REGION Network 9: fDoor5 monitoring
   RUNG wire#powerrail
      Contact( #TRUE )
      wire#w1
      Contact( "Safety.DataFromSafety".fDoorCoilStatus.weightNgBoxDoorUnlock )
      wire#w2
      Coil( "SafetyDoorInterface".fDoor5Interface.monitoring.DoorOpen )
   END_RUNG
   RUNG wire#w1
      I_Contact( "Safety.DataFromSafety".fDoorCoilStatus.weightNgBoxDoorUnlock )
      Contact( "Safety.DataFromSafety".fDoorDrive.fDoor5.ackReq )
      I_Contact( "Global.Data".general.clock.cycle1000Msec )
      I_Contact( "Safety.DataFromSafety".fDoorSwitchStatus.weightNgBoxDoorOpen )
   END_RUNG wire#w2
   RUNG wire#w1
      Contact( "Safety.DataFromSafety".fDoorCoilStatus.weightNgBoxDoorUnlock )
      Coil( "SafetyDoorInterface".fDoor5Interface.monitoring.DoorUnLock )
   END_RUNG
   RUNG wire#w1
      I_Contact( "Safety.DataFromSafety".fDoorCoilStatus.weightNgBoxDoorUnlock )
      wire#w3
      I_Contact( "Safety.DataFromSafety".fDoorDrive.fDoor5.ackReq )
      wire#w4
      I_Contact( "Safety.DataFromSafety".fDoorSwitchStatus.weightNgBoxDoorOpen )
      I_Contact( "SafetyDoorInterface".fDoor5Interface.monitoring.DoorOpen )
      Coil( "SafetyDoorInterface".fDoor5Interface.monitoring.DoorClose )
   END_RUNG
   RUNG wire#w3
      Contact( "Safety.DataFromSafety".fDoorDrive.fDoor5.ackReq )
      I_Contact( "Global.Data".general.clock.cycle1000Msec )
   END_RUNG wire#w4
   RUNG wire#w4
      Coil( "SafetyDoorInterface".fDoor5Interface.monitoring.DoorLock )
   END_RUNG
   // the same network as SCL:
   "SafetyDoorInterface".fDoor5Interface.monitoring.DoorOpen := #TRUE AND ("Safety.DataFromSafety".fDoorCoilStatus.weightNgBoxDoorUnlock OR (NOT "Safety.DataFromSafety".fDoorCoilStatus.weightNgBoxDoorUnlock AND "Safety.DataFromSafety".fDoorDrive.fDoor5.ackReq AND NOT "Global.Data".general.clock.cycle1000Msec AND NOT "Safety.DataFromSafety".fDoorSwitchStatus.weightNgBoxDoorOpen));
   "SafetyDoorInterface".fDoor5Interface.monitoring.DoorUnLock := #TRUE AND "Safety.DataFromSafety".fDoorCoilStatus.weightNgBoxDoorUnlock;
   #_w1 := #TRUE AND NOT "Safety.DataFromSafety".fDoorCoilStatus.weightNgBoxDoorUnlock AND (NOT "Safety.DataFromSafety".fDoorDrive.fDoor5.ackReq OR ("Safety.DataFromSafety".fDoorDrive.fDoor5.ackReq AND NOT "Global.Data".general.clock.cycle1000Msec));
   "SafetyDoorInterface".fDoor5Interface.monitoring.DoorClose := #_w1 AND NOT "Safety.DataFromSafety".fDoorSwitchStatus.weightNgBoxDoorOpen AND NOT "SafetyDoorInterface".fDoor5Interface.monitoring.DoorOpen;
   "SafetyDoorInterface".fDoor5Interface.monitoring.DoorLock := #_w1;
END_REGION

REGION Network 10: fDoor5 Command
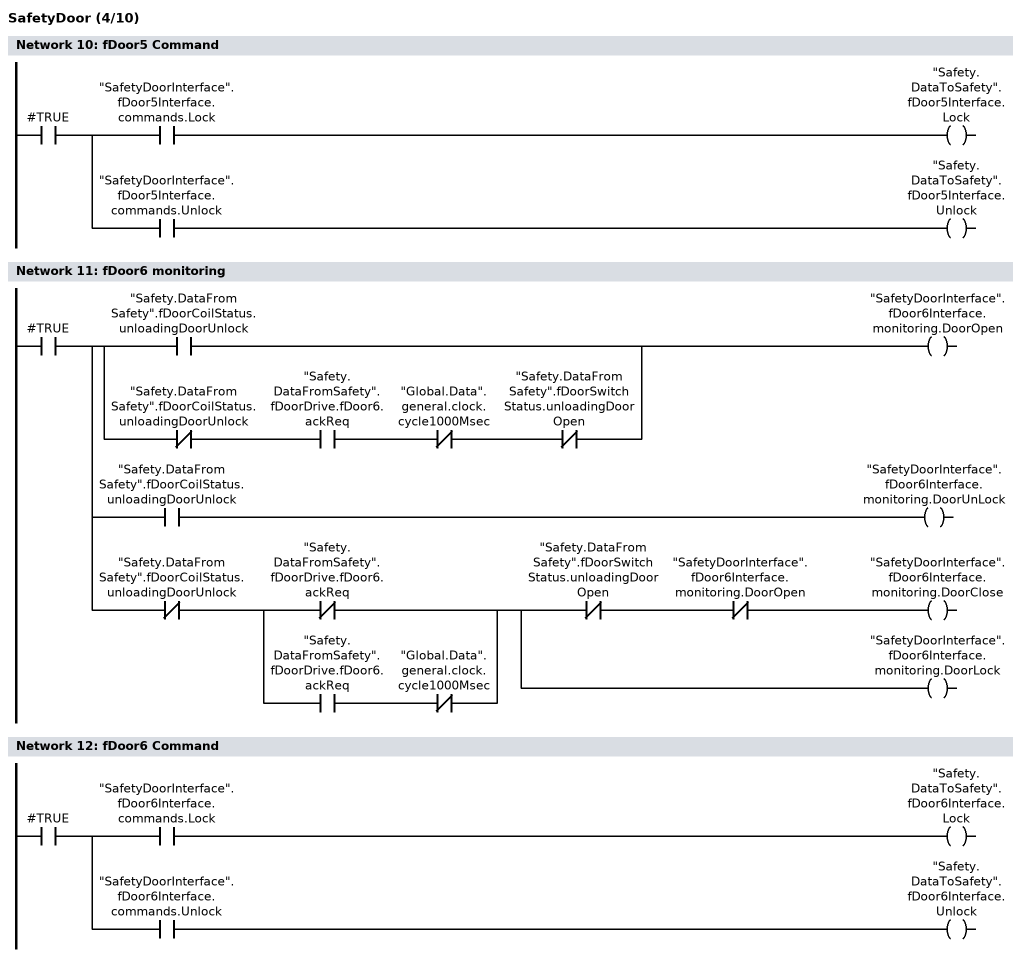
   RUNG wire#powerrail
      Contact( #TRUE )
      wire#w1
      Contact( "SafetyDoorInterface".fDoor5Interface.commands.Lock )
      Coil( "Safety.DataToSafety".fDoor5Interface.Lock )
   END_RUNG
   RUNG wire#w1
      Contact( "SafetyDoorInterface".fDoor5Interface.commands.Unlock )
      Coil( "Safety.DataToSafety".fDoor5Interface.Unlock )
   END_RUNG
   // the same network as SCL:
   "Safety.DataToSafety".fDoor5Interface.Lock := #TRUE AND "SafetyDoorInterface".fDoor5Interface.commands.Lock;
   "Safety.DataToSafety".fDoor5Interface.Unlock := #TRUE AND "SafetyDoorInterface".fDoor5Interface.commands.Unlock;
END_REGION

REGION Network 11: fDoor6 monitoring
   RUNG wire#powerrail
      Contact( #TRUE )
      wire#w1
      Contact( "Safety.DataFromSafety".fDoorCoilStatus.unloadingDoorUnlock )
      wire#w2
      Coil( "SafetyDoorInterface".fDoor6Interface.monitoring.DoorOpen )
   END_RUNG
   RUNG wire#w1
      I_Contact( "Safety.DataFromSafety".fDoorCoilStatus.unloadingDoorUnlock )
      Contact( "Safety.DataFromSafety".fDoorDrive.fDoor6.ackReq )
      I_Contact( "Global.Data".general.clock.cycle1000Msec )
      I_Contact( "Safety.DataFromSafety".fDoorSwitchStatus.unloadingDoorOpen )
   END_RUNG wire#w2
   RUNG wire#w1
      Contact( "Safety.DataFromSafety".fDoorCoilStatus.unloadingDoorUnlock )
      Coil( "SafetyDoorInterface".fDoor6Interface.monitoring.DoorUnLock )
   END_RUNG
   RUNG wire#w1
      I_Contact( "Safety.DataFromSafety".fDoorCoilStatus.unloadingDoorUnlock )
      wire#w3
      I_Contact( "Safety.DataFromSafety".fDoorDrive.fDoor6.ackReq )
      wire#w4
      I_Contact( "Safety.DataFromSafety".fDoorSwitchStatus.unloadingDoorOpen )
      I_Contact( "SafetyDoorInterface".fDoor6Interface.monitoring.DoorOpen )
      Coil( "SafetyDoorInterface".fDoor6Interface.monitoring.DoorClose )
   END_RUNG
   RUNG wire#w3
      Contact( "Safety.DataFromSafety".fDoorDrive.fDoor6.ackReq )
      I_Contact( "Global.Data".general.clock.cycle1000Msec )
   END_RUNG wire#w4
   RUNG wire#w4
      Coil( "SafetyDoorInterface".fDoor6Interface.monitoring.DoorLock )
   END_RUNG
   // the same network as SCL:
   "SafetyDoorInterface".fDoor6Interface.monitoring.DoorOpen := #TRUE AND ("Safety.DataFromSafety".fDoorCoilStatus.unloadingDoorUnlock OR (NOT "Safety.DataFromSafety".fDoorCoilStatus.unloadingDoorUnlock AND "Safety.DataFromSafety".fDoorDrive.fDoor6.ackReq AND NOT "Global.Data".general.clock.cycle1000Msec AND NOT "Safety.DataFromSafety".fDoorSwitchStatus.unloadingDoorOpen));
   "SafetyDoorInterface".fDoor6Interface.monitoring.DoorUnLock := #TRUE AND "Safety.DataFromSafety".fDoorCoilStatus.unloadingDoorUnlock;
   #_w1 := #TRUE AND NOT "Safety.DataFromSafety".fDoorCoilStatus.unloadingDoorUnlock AND (NOT "Safety.DataFromSafety".fDoorDrive.fDoor6.ackReq OR ("Safety.DataFromSafety".fDoorDrive.fDoor6.ackReq AND NOT "Global.Data".general.clock.cycle1000Msec));
   "SafetyDoorInterface".fDoor6Interface.monitoring.DoorClose := #_w1 AND NOT "Safety.DataFromSafety".fDoorSwitchStatus.unloadingDoorOpen AND NOT "SafetyDoorInterface".fDoor6Interface.monitoring.DoorOpen;
   "SafetyDoorInterface".fDoor6Interface.monitoring.DoorLock := #_w1;
END_REGION

REGION Network 12: fDoor6 Command
   RUNG wire#powerrail
      Contact( #TRUE )
      wire#w1
      Contact( "SafetyDoorInterface".fDoor6Interface.commands.Lock )
      Coil( "Safety.DataToSafety".fDoor6Interface.Lock )
   END_RUNG
   RUNG wire#w1
      Contact( "SafetyDoorInterface".fDoor6Interface.commands.Unlock )
      Coil( "Safety.DataToSafety".fDoor6Interface.Unlock )
   END_RUNG
   // the same network as SCL:
   "Safety.DataToSafety".fDoor6Interface.Lock := #TRUE AND "SafetyDoorInterface".fDoor6Interface.commands.Lock;
   "Safety.DataToSafety".fDoor6Interface.Unlock := #TRUE AND "SafetyDoorInterface".fDoor6Interface.commands.Unlock;
END_REGION

REGION Network 13: fDoor7 monitoring
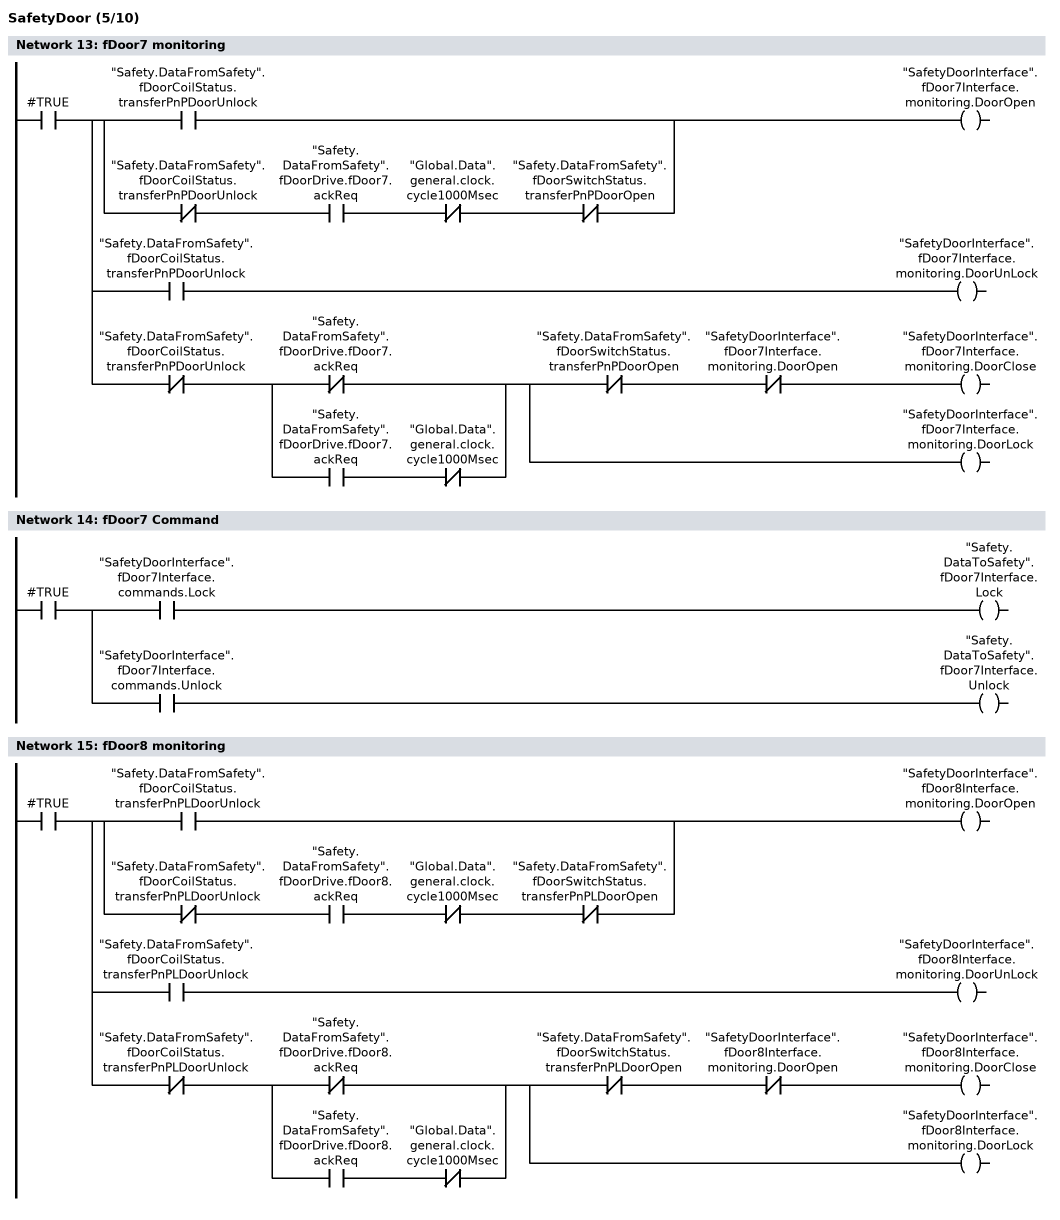
   RUNG wire#powerrail
      Contact( #TRUE )
      wire#w1
      Contact( "Safety.DataFromSafety".fDoorCoilStatus.transferPnPDoorUnlock )
      wire#w2
      Coil( "SafetyDoorInterface".fDoor7Interface.monitoring.DoorOpen )
   END_RUNG
   RUNG wire#w1
      I_Contact( "Safety.DataFromSafety".fDoorCoilStatus.transferPnPDoorUnlock )
      Contact( "Safety.DataFromSafety".fDoorDrive.fDoor7.ackReq )
      I_Contact( "Global.Data".general.clock.cycle1000Msec )
      I_Contact( "Safety.DataFromSafety".fDoorSwitchStatus.transferPnPDoorOpen )
   END_RUNG wire#w2
   RUNG wire#w1
      Contact( "Safety.DataFromSafety".fDoorCoilStatus.transferPnPDoorUnlock )
      Coil( "SafetyDoorInterface".fDoor7Interface.monitoring.DoorUnLock )
   END_RUNG
   RUNG wire#w1
      I_Contact( "Safety.DataFromSafety".fDoorCoilStatus.transferPnPDoorUnlock )
      wire#w3
      I_Contact( "Safety.DataFromSafety".fDoorDrive.fDoor7.ackReq )
      wire#w4
      I_Contact( "Safety.DataFromSafety".fDoorSwitchStatus.transferPnPDoorOpen )
      I_Contact( "SafetyDoorInterface".fDoor7Interface.monitoring.DoorOpen )
      Coil( "SafetyDoorInterface".fDoor7Interface.monitoring.DoorClose )
   END_RUNG
   RUNG wire#w3
      Contact( "Safety.DataFromSafety".fDoorDrive.fDoor7.ackReq )
      I_Contact( "Global.Data".general.clock.cycle1000Msec )
   END_RUNG wire#w4
   RUNG wire#w4
      Coil( "SafetyDoorInterface".fDoor7Interface.monitoring.DoorLock )
   END_RUNG
   // the same network as SCL:
   "SafetyDoorInterface".fDoor7Interface.monitoring.DoorOpen := #TRUE AND ("Safety.DataFromSafety".fDoorCoilStatus.transferPnPDoorUnlock OR (NOT "Safety.DataFromSafety".fDoorCoilStatus.transferPnPDoorUnlock AND "Safety.DataFromSafety".fDoorDrive.fDoor7.ackReq AND NOT "Global.Data".general.clock.cycle1000Msec AND NOT "Safety.DataFromSafety".fDoorSwitchStatus.transferPnPDoorOpen));
   "SafetyDoorInterface".fDoor7Interface.monitoring.DoorUnLock := #TRUE AND "Safety.DataFromSafety".fDoorCoilStatus.transferPnPDoorUnlock;
   #_w1 := #TRUE AND NOT "Safety.DataFromSafety".fDoorCoilStatus.transferPnPDoorUnlock AND (NOT "Safety.DataFromSafety".fDoorDrive.fDoor7.ackReq OR ("Safety.DataFromSafety".fDoorDrive.fDoor7.ackReq AND NOT "Global.Data".general.clock.cycle1000Msec));
   "SafetyDoorInterface".fDoor7Interface.monitoring.DoorClose := #_w1 AND NOT "Safety.DataFromSafety".fDoorSwitchStatus.transferPnPDoorOpen AND NOT "SafetyDoorInterface".fDoor7Interface.monitoring.DoorOpen;
   "SafetyDoorInterface".fDoor7Interface.monitoring.DoorLock := #_w1;
END_REGION

REGION Network 14: fDoor7 Command
   RUNG wire#powerrail
      Contact( #TRUE )
      wire#w1
      Contact( "SafetyDoorInterface".fDoor7Interface.commands.Lock )
      Coil( "Safety.DataToSafety".fDoor7Interface.Lock )
   END_RUNG
   RUNG wire#w1
      Contact( "SafetyDoorInterface".fDoor7Interface.commands.Unlock )
      Coil( "Safety.DataToSafety".fDoor7Interface.Unlock )
   END_RUNG
   // the same network as SCL:
   "Safety.DataToSafety".fDoor7Interface.Lock := #TRUE AND "SafetyDoorInterface".fDoor7Interface.commands.Lock;
   "Safety.DataToSafety".fDoor7Interface.Unlock := #TRUE AND "SafetyDoorInterface".fDoor7Interface.commands.Unlock;
END_REGION

REGION Network 15: fDoor8 monitoring
   RUNG wire#powerrail
      Contact( #TRUE )
      wire#w1
      Contact( "Safety.DataFromSafety".fDoorCoilStatus.transferPnPLDoorUnlock )
      wire#w2
      Coil( "SafetyDoorInterface".fDoor8Interface.monitoring.DoorOpen )
   END_RUNG
   RUNG wire#w1
      I_Contact( "Safety.DataFromSafety".fDoorCoilStatus.transferPnPLDoorUnlock )
      Contact( "Safety.DataFromSafety".fDoorDrive.fDoor8.ackReq )
      I_Contact( "Global.Data".general.clock.cycle1000Msec )
      I_Contact( "Safety.DataFromSafety".fDoorSwitchStatus.transferPnPLDoorOpen )
   END_RUNG wire#w2
   RUNG wire#w1
      Contact( "Safety.DataFromSafety".fDoorCoilStatus.transferPnPLDoorUnlock )
      Coil( "SafetyDoorInterface".fDoor8Interface.monitoring.DoorUnLock )
   END_RUNG
   RUNG wire#w1
      I_Contact( "Safety.DataFromSafety".fDoorCoilStatus.transferPnPLDoorUnlock )
      wire#w3
      I_Contact( "Safety.DataFromSafety".fDoorDrive.fDoor8.ackReq )
      wire#w4
      I_Contact( "Safety.DataFromSafety".fDoorSwitchStatus.transferPnPLDoorOpen )
      I_Contact( "SafetyDoorInterface".fDoor8Interface.monitoring.DoorOpen )
      Coil( "SafetyDoorInterface".fDoor8Interface.monitoring.DoorClose )
   END_RUNG
   RUNG wire#w3
      Contact( "Safety.DataFromSafety".fDoorDrive.fDoor8.ackReq )
      I_Contact( "Global.Data".general.clock.cycle1000Msec )
   END_RUNG wire#w4
   RUNG wire#w4
      Coil( "SafetyDoorInterface".fDoor8Interface.monitoring.DoorLock )
   END_RUNG
   // the same network as SCL:
   "SafetyDoorInterface".fDoor8Interface.monitoring.DoorOpen := #TRUE AND ("Safety.DataFromSafety".fDoorCoilStatus.transferPnPLDoorUnlock OR (NOT "Safety.DataFromSafety".fDoorCoilStatus.transferPnPLDoorUnlock AND "Safety.DataFromSafety".fDoorDrive.fDoor8.ackReq AND NOT "Global.Data".general.clock.cycle1000Msec AND NOT "Safety.DataFromSafety".fDoorSwitchStatus.transferPnPLDoorOpen));
   "SafetyDoorInterface".fDoor8Interface.monitoring.DoorUnLock := #TRUE AND "Safety.DataFromSafety".fDoorCoilStatus.transferPnPLDoorUnlock;
   #_w1 := #TRUE AND NOT "Safety.DataFromSafety".fDoorCoilStatus.transferPnPLDoorUnlock AND (NOT "Safety.DataFromSafety".fDoorDrive.fDoor8.ackReq OR ("Safety.DataFromSafety".fDoorDrive.fDoor8.ackReq AND NOT "Global.Data".general.clock.cycle1000Msec));
   "SafetyDoorInterface".fDoor8Interface.monitoring.DoorClose := #_w1 AND NOT "Safety.DataFromSafety".fDoorSwitchStatus.transferPnPLDoorOpen AND NOT "SafetyDoorInterface".fDoor8Interface.monitoring.DoorOpen;
   "SafetyDoorInterface".fDoor8Interface.monitoring.DoorLock := #_w1;
END_REGION

REGION Network 16: fDoor8 Command
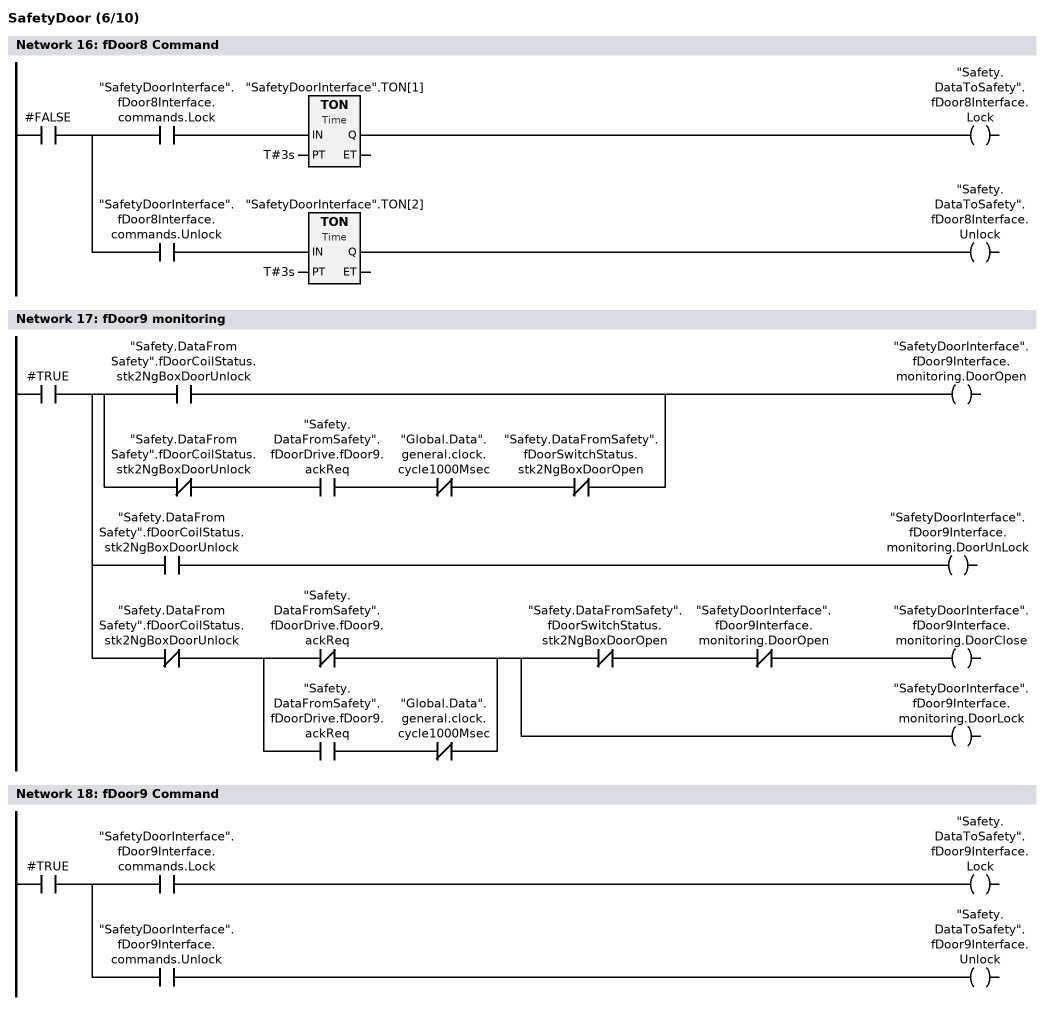
   RUNG wire#powerrail
      Contact( #FALSE )
      wire#w1
      Contact( "SafetyDoorInterface".fDoor8Interface.commands.Lock )
      { S7_Templates := "time_type := Time" } "SafetyDoorInterface".TON[1].TON(pt := T#3s, et =>)
      Coil( "Safety.DataToSafety".fDoor8Interface.Lock )
   END_RUNG
   RUNG wire#w1
      Contact( "SafetyDoorInterface".fDoor8Interface.commands.Unlock )
      { S7_Templates := "time_type := Time" } "SafetyDoorInterface".TON[2].TON(pt := T#3s, et =>)
      Coil( "Safety.DataToSafety".fDoor8Interface.Unlock )
   END_RUNG
   // the same network as SCL:
   "SafetyDoorInterface".TON[1].TON(IN := #FALSE AND "SafetyDoorInterface".fDoor8Interface.commands.Lock,
                           PT := T#3s);
   "Safety.DataToSafety".fDoor8Interface.Lock := "SafetyDoorInterface".TON[1].Q;
   "SafetyDoorInterface".TON[2].TON(IN := #FALSE AND "SafetyDoorInterface".fDoor8Interface.commands.Unlock,
                           PT := T#3s);
   "Safety.DataToSafety".fDoor8Interface.Unlock := "SafetyDoorInterface".TON[2].Q;
END_REGION

REGION Network 17: fDoor9 monitoring
   RUNG wire#powerrail
      Contact( #TRUE )
      wire#w1
      Contact( "Safety.DataFromSafety".fDoorCoilStatus.stk2NgBoxDoorUnlock )
      wire#w2
      Coil( "SafetyDoorInterface".fDoor9Interface.monitoring.DoorOpen )
   END_RUNG
   RUNG wire#w1
      I_Contact( "Safety.DataFromSafety".fDoorCoilStatus.stk2NgBoxDoorUnlock )
      Contact( "Safety.DataFromSafety".fDoorDrive.fDoor9.ackReq )
      I_Contact( "Global.Data".general.clock.cycle1000Msec )
      I_Contact( "Safety.DataFromSafety".fDoorSwitchStatus.stk2NgBoxDoorOpen )
   END_RUNG wire#w2
   RUNG wire#w1
      Contact( "Safety.DataFromSafety".fDoorCoilStatus.stk2NgBoxDoorUnlock )
      Coil( "SafetyDoorInterface".fDoor9Interface.monitoring.DoorUnLock )
   END_RUNG
   RUNG wire#w1
      I_Contact( "Safety.DataFromSafety".fDoorCoilStatus.stk2NgBoxDoorUnlock )
      wire#w3
      I_Contact( "Safety.DataFromSafety".fDoorDrive.fDoor9.ackReq )
      wire#w4
      I_Contact( "Safety.DataFromSafety".fDoorSwitchStatus.stk2NgBoxDoorOpen )
      I_Contact( "SafetyDoorInterface".fDoor9Interface.monitoring.DoorOpen )
      Coil( "SafetyDoorInterface".fDoor9Interface.monitoring.DoorClose )
   END_RUNG
   RUNG wire#w3
      Contact( "Safety.DataFromSafety".fDoorDrive.fDoor9.ackReq )
      I_Contact( "Global.Data".general.clock.cycle1000Msec )
   END_RUNG wire#w4
   RUNG wire#w4
      Coil( "SafetyDoorInterface".fDoor9Interface.monitoring.DoorLock )
   END_RUNG
   // the same network as SCL:
   "SafetyDoorInterface".fDoor9Interface.monitoring.DoorOpen := #TRUE AND ("Safety.DataFromSafety".fDoorCoilStatus.stk2NgBoxDoorUnlock OR (NOT "Safety.DataFromSafety".fDoorCoilStatus.stk2NgBoxDoorUnlock AND "Safety.DataFromSafety".fDoorDrive.fDoor9.ackReq AND NOT "Global.Data".general.clock.cycle1000Msec AND NOT "Safety.DataFromSafety".fDoorSwitchStatus.stk2NgBoxDoorOpen));
   "SafetyDoorInterface".fDoor9Interface.monitoring.DoorUnLock := #TRUE AND "Safety.DataFromSafety".fDoorCoilStatus.stk2NgBoxDoorUnlock;
   #_w1 := #TRUE AND NOT "Safety.DataFromSafety".fDoorCoilStatus.stk2NgBoxDoorUnlock AND (NOT "Safety.DataFromSafety".fDoorDrive.fDoor9.ackReq OR ("Safety.DataFromSafety".fDoorDrive.fDoor9.ackReq AND NOT "Global.Data".general.clock.cycle1000Msec));
   "SafetyDoorInterface".fDoor9Interface.monitoring.DoorClose := #_w1 AND NOT "Safety.DataFromSafety".fDoorSwitchStatus.stk2NgBoxDoorOpen AND NOT "SafetyDoorInterface".fDoor9Interface.monitoring.DoorOpen;
   "SafetyDoorInterface".fDoor9Interface.monitoring.DoorLock := #_w1;
END_REGION

REGION Network 18: fDoor9 Command
   RUNG wire#powerrail
      Contact( #TRUE )
      wire#w1
      Contact( "SafetyDoorInterface".fDoor9Interface.commands.Lock )
      Coil( "Safety.DataToSafety".fDoor9Interface.Lock )
   END_RUNG
   RUNG wire#w1
      Contact( "SafetyDoorInterface".fDoor9Interface.commands.Unlock )
      Coil( "Safety.DataToSafety".fDoor9Interface.Unlock )
   END_RUNG
   // the same network as SCL:
   "Safety.DataToSafety".fDoor9Interface.Lock := #TRUE AND "SafetyDoorInterface".fDoor9Interface.commands.Lock;
   "Safety.DataToSafety".fDoor9Interface.Unlock := #TRUE AND "SafetyDoorInterface".fDoor9Interface.commands.Unlock;
END_REGION

REGION Network 19: fDoor10 monitoring
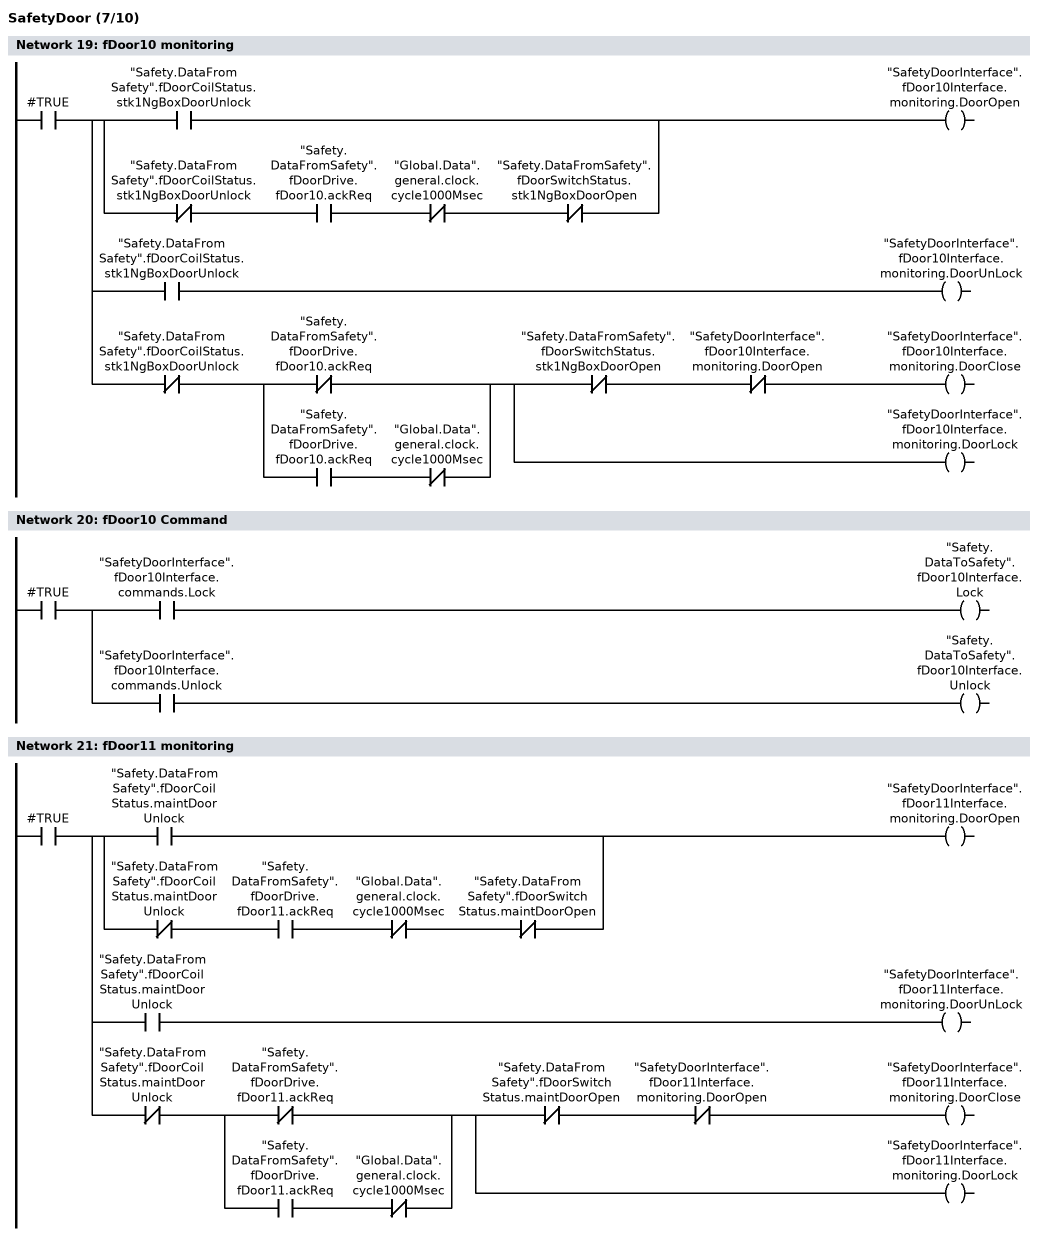
   RUNG wire#powerrail
      Contact( #TRUE )
      wire#w1
      Contact( "Safety.DataFromSafety".fDoorCoilStatus.stk1NgBoxDoorUnlock )
      wire#w2
      Coil( "SafetyDoorInterface".fDoor10Interface.monitoring.DoorOpen )
   END_RUNG
   RUNG wire#w1
      I_Contact( "Safety.DataFromSafety".fDoorCoilStatus.stk1NgBoxDoorUnlock )
      Contact( "Safety.DataFromSafety".fDoorDrive.fDoor10.ackReq )
      I_Contact( "Global.Data".general.clock.cycle1000Msec )
      I_Contact( "Safety.DataFromSafety".fDoorSwitchStatus.stk1NgBoxDoorOpen )
   END_RUNG wire#w2
   RUNG wire#w1
      Contact( "Safety.DataFromSafety".fDoorCoilStatus.stk1NgBoxDoorUnlock )
      Coil( "SafetyDoorInterface".fDoor10Interface.monitoring.DoorUnLock )
   END_RUNG
   RUNG wire#w1
      I_Contact( "Safety.DataFromSafety".fDoorCoilStatus.stk1NgBoxDoorUnlock )
      wire#w3
      I_Contact( "Safety.DataFromSafety".fDoorDrive.fDoor10.ackReq )
      wire#w4
      I_Contact( "Safety.DataFromSafety".fDoorSwitchStatus.stk1NgBoxDoorOpen )
      I_Contact( "SafetyDoorInterface".fDoor10Interface.monitoring.DoorOpen )
      Coil( "SafetyDoorInterface".fDoor10Interface.monitoring.DoorClose )
   END_RUNG
   RUNG wire#w3
      Contact( "Safety.DataFromSafety".fDoorDrive.fDoor10.ackReq )
      I_Contact( "Global.Data".general.clock.cycle1000Msec )
   END_RUNG wire#w4
   RUNG wire#w4
      Coil( "SafetyDoorInterface".fDoor10Interface.monitoring.DoorLock )
   END_RUNG
   // the same network as SCL:
   "SafetyDoorInterface".fDoor10Interface.monitoring.DoorOpen := #TRUE AND ("Safety.DataFromSafety".fDoorCoilStatus.stk1NgBoxDoorUnlock OR (NOT "Safety.DataFromSafety".fDoorCoilStatus.stk1NgBoxDoorUnlock AND "Safety.DataFromSafety".fDoorDrive.fDoor10.ackReq AND NOT "Global.Data".general.clock.cycle1000Msec AND NOT "Safety.DataFromSafety".fDoorSwitchStatus.stk1NgBoxDoorOpen));
   "SafetyDoorInterface".fDoor10Interface.monitoring.DoorUnLock := #TRUE AND "Safety.DataFromSafety".fDoorCoilStatus.stk1NgBoxDoorUnlock;
   #_w1 := #TRUE AND NOT "Safety.DataFromSafety".fDoorCoilStatus.stk1NgBoxDoorUnlock AND (NOT "Safety.DataFromSafety".fDoorDrive.fDoor10.ackReq OR ("Safety.DataFromSafety".fDoorDrive.fDoor10.ackReq AND NOT "Global.Data".general.clock.cycle1000Msec));
   "SafetyDoorInterface".fDoor10Interface.monitoring.DoorClose := #_w1 AND NOT "Safety.DataFromSafety".fDoorSwitchStatus.stk1NgBoxDoorOpen AND NOT "SafetyDoorInterface".fDoor10Interface.monitoring.DoorOpen;
   "SafetyDoorInterface".fDoor10Interface.monitoring.DoorLock := #_w1;
END_REGION

REGION Network 20: fDoor10 Command
   RUNG wire#powerrail
      Contact( #TRUE )
      wire#w1
      Contact( "SafetyDoorInterface".fDoor10Interface.commands.Lock )
      Coil( "Safety.DataToSafety".fDoor10Interface.Lock )
   END_RUNG
   RUNG wire#w1
      Contact( "SafetyDoorInterface".fDoor10Interface.commands.Unlock )
      Coil( "Safety.DataToSafety".fDoor10Interface.Unlock )
   END_RUNG
   // the same network as SCL:
   "Safety.DataToSafety".fDoor10Interface.Lock := #TRUE AND "SafetyDoorInterface".fDoor10Interface.commands.Lock;
   "Safety.DataToSafety".fDoor10Interface.Unlock := #TRUE AND "SafetyDoorInterface".fDoor10Interface.commands.Unlock;
END_REGION

REGION Network 21: fDoor11 monitoring
   RUNG wire#powerrail
      Contact( #TRUE )
      wire#w1
      Contact( "Safety.DataFromSafety".fDoorCoilStatus.maintDoorUnlock )
      wire#w2
      Coil( "SafetyDoorInterface".fDoor11Interface.monitoring.DoorOpen )
   END_RUNG
   RUNG wire#w1
      I_Contact( "Safety.DataFromSafety".fDoorCoilStatus.maintDoorUnlock )
      Contact( "Safety.DataFromSafety".fDoorDrive.fDoor11.ackReq )
      I_Contact( "Global.Data".general.clock.cycle1000Msec )
      I_Contact( "Safety.DataFromSafety".fDoorSwitchStatus.maintDoorOpen )
   END_RUNG wire#w2
   RUNG wire#w1
      Contact( "Safety.DataFromSafety".fDoorCoilStatus.maintDoorUnlock )
      Coil( "SafetyDoorInterface".fDoor11Interface.monitoring.DoorUnLock )
   END_RUNG
   RUNG wire#w1
      I_Contact( "Safety.DataFromSafety".fDoorCoilStatus.maintDoorUnlock )
      wire#w3
      I_Contact( "Safety.DataFromSafety".fDoorDrive.fDoor11.ackReq )
      wire#w4
      I_Contact( "Safety.DataFromSafety".fDoorSwitchStatus.maintDoorOpen )
      I_Contact( "SafetyDoorInterface".fDoor11Interface.monitoring.DoorOpen )
      Coil( "SafetyDoorInterface".fDoor11Interface.monitoring.DoorClose )
   END_RUNG
   RUNG wire#w3
      Contact( "Safety.DataFromSafety".fDoorDrive.fDoor11.ackReq )
      I_Contact( "Global.Data".general.clock.cycle1000Msec )
   END_RUNG wire#w4
   RUNG wire#w4
      Coil( "SafetyDoorInterface".fDoor11Interface.monitoring.DoorLock )
   END_RUNG
   // the same network as SCL:
   "SafetyDoorInterface".fDoor11Interface.monitoring.DoorOpen := #TRUE AND ("Safety.DataFromSafety".fDoorCoilStatus.maintDoorUnlock OR (NOT "Safety.DataFromSafety".fDoorCoilStatus.maintDoorUnlock AND "Safety.DataFromSafety".fDoorDrive.fDoor11.ackReq AND NOT "Global.Data".general.clock.cycle1000Msec AND NOT "Safety.DataFromSafety".fDoorSwitchStatus.maintDoorOpen));
   "SafetyDoorInterface".fDoor11Interface.monitoring.DoorUnLock := #TRUE AND "Safety.DataFromSafety".fDoorCoilStatus.maintDoorUnlock;
   #_w1 := #TRUE AND NOT "Safety.DataFromSafety".fDoorCoilStatus.maintDoorUnlock AND (NOT "Safety.DataFromSafety".fDoorDrive.fDoor11.ackReq OR ("Safety.DataFromSafety".fDoorDrive.fDoor11.ackReq AND NOT "Global.Data".general.clock.cycle1000Msec));
   "SafetyDoorInterface".fDoor11Interface.monitoring.DoorClose := #_w1 AND NOT "Safety.DataFromSafety".fDoorSwitchStatus.maintDoorOpen AND NOT "SafetyDoorInterface".fDoor11Interface.monitoring.DoorOpen;
   "SafetyDoorInterface".fDoor11Interface.monitoring.DoorLock := #_w1;
END_REGION

REGION Network 22: fDoor11 Command
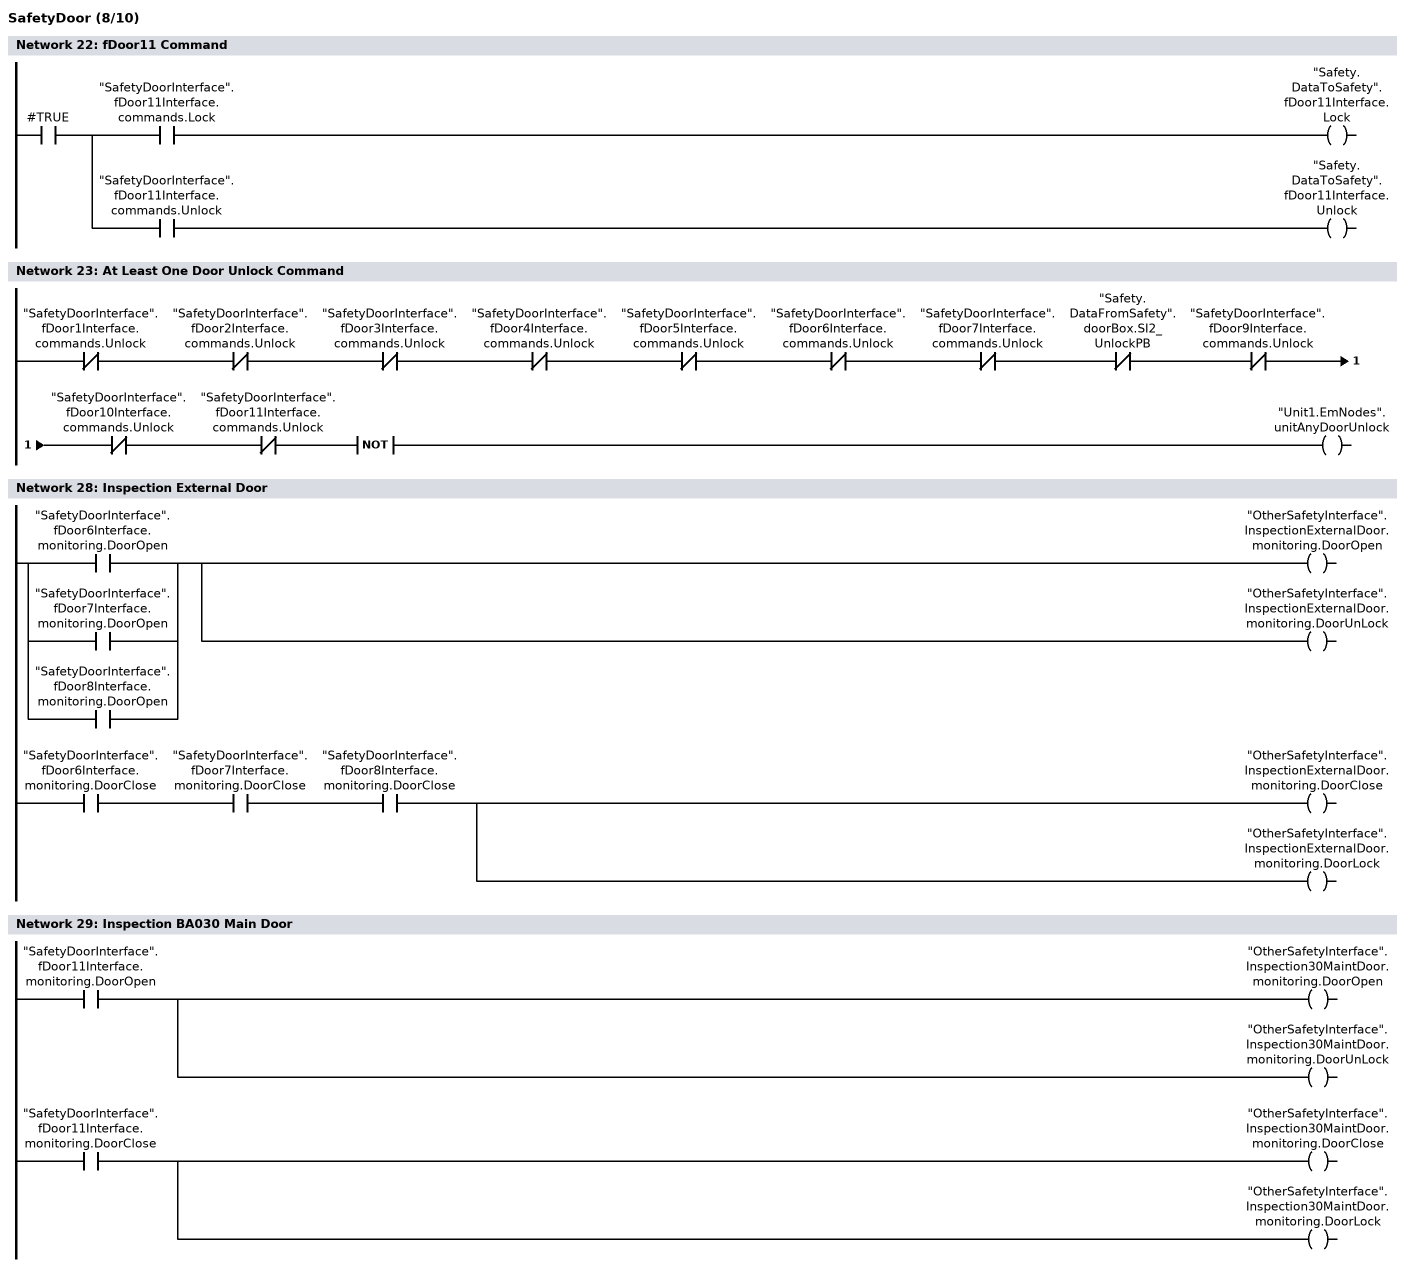
   RUNG wire#powerrail
      Contact( #TRUE )
      wire#w1
      Contact( "SafetyDoorInterface".fDoor11Interface.commands.Lock )
      Coil( "Safety.DataToSafety".fDoor11Interface.Lock )
   END_RUNG
   RUNG wire#w1
      Contact( "SafetyDoorInterface".fDoor11Interface.commands.Unlock )
      Coil( "Safety.DataToSafety".fDoor11Interface.Unlock )
   END_RUNG
   // the same network as SCL:
   "Safety.DataToSafety".fDoor11Interface.Lock := #TRUE AND "SafetyDoorInterface".fDoor11Interface.commands.Lock;
   "Safety.DataToSafety".fDoor11Interface.Unlock := #TRUE AND "SafetyDoorInterface".fDoor11Interface.commands.Unlock;
END_REGION

REGION Network 23: At Least One Door Unlock Command
   RUNG wire#powerrail
      I_Contact( "SafetyDoorInterface".fDoor1Interface.commands.Unlock )
      I_Contact( "SafetyDoorInterface".fDoor2Interface.commands.Unlock )
      I_Contact( "SafetyDoorInterface".fDoor3Interface.commands.Unlock )
      I_Contact( "SafetyDoorInterface".fDoor4Interface.commands.Unlock )
      I_Contact( "SafetyDoorInterface".fDoor5Interface.commands.Unlock )
      I_Contact( "SafetyDoorInterface".fDoor6Interface.commands.Unlock )
      I_Contact( "SafetyDoorInterface".fDoor7Interface.commands.Unlock )
      I_Contact( "Safety.DataFromSafety".doorBox.SI2_UnlockPB )
      I_Contact( "SafetyDoorInterface".fDoor9Interface.commands.Unlock )
      I_Contact( "SafetyDoorInterface".fDoor10Interface.commands.Unlock )
      I_Contact( "SafetyDoorInterface".fDoor11Interface.commands.Unlock )
      Not()
      Coil( "Unit1.EmNodes".unitAnyDoorUnlock )
   END_RUNG
   // the same network as SCL:
   "Unit1.EmNodes".unitAnyDoorUnlock := NOT (NOT "SafetyDoorInterface".fDoor1Interface.commands.Unlock AND NOT "SafetyDoorInterface".fDoor2Interface.commands.Unlock AND NOT "SafetyDoorInterface".fDoor3Interface.commands.Unlock AND NOT "SafetyDoorInterface".fDoor4Interface.commands.Unlock AND NOT "SafetyDoorInterface".fDoor5Interface.commands.Unlock AND NOT "SafetyDoorInterface".fDoor6Interface.commands.Unlock AND NOT "SafetyDoorInterface".fDoor7Interface.commands.Unlock AND NOT "Safety.DataFromSafety".doorBox.SI2_UnlockPB AND NOT "SafetyDoorInterface".fDoor9Interface.commands.Unlock AND NOT "SafetyDoorInterface".fDoor10Interface.commands.Unlock AND NOT "SafetyDoorInterface".fDoor11Interface.commands.Unlock);
END_REGION

REGION Network 24: BA010 Other Door
END_REGION

REGION Network 25: BA015 Other Door
END_REGION

REGION Network 26: BA030 Other Door
END_REGION

REGION Network 27: BA040 Other Door
END_REGION

REGION Network 28: Inspection External Door
   RUNG wire#powerrail
      Contact( "SafetyDoorInterface".fDoor6Interface.monitoring.DoorOpen )
      wire#w1
      Coil( "OtherSafetyInterface".InspectionExternalDoor.monitoring.DoorOpen )
   END_RUNG
   RUNG wire#powerrail
      Contact( "SafetyDoorInterface".fDoor7Interface.monitoring.DoorOpen )
   END_RUNG wire#w1
   RUNG wire#powerrail
      Contact( "SafetyDoorInterface".fDoor8Interface.monitoring.DoorOpen )
   END_RUNG wire#w1
   RUNG wire#w1
      Coil( "OtherSafetyInterface".InspectionExternalDoor.monitoring.DoorUnLock )
   END_RUNG
   RUNG wire#powerrail
      Contact( "SafetyDoorInterface".fDoor6Interface.monitoring.DoorClose )
      Contact( "SafetyDoorInterface".fDoor7Interface.monitoring.DoorClose )
      Contact( "SafetyDoorInterface".fDoor8Interface.monitoring.DoorClose )
      wire#w2
      Coil( "OtherSafetyInterface".InspectionExternalDoor.monitoring.DoorClose )
   END_RUNG
   RUNG wire#w2
      Coil( "OtherSafetyInterface".InspectionExternalDoor.monitoring.DoorLock )
   END_RUNG
   // the same network as SCL:
   "OtherSafetyInterface".InspectionExternalDoor.monitoring.DoorOpen := "SafetyDoorInterface".fDoor6Interface.monitoring.DoorOpen OR "SafetyDoorInterface".fDoor7Interface.monitoring.DoorOpen OR "SafetyDoorInterface".fDoor8Interface.monitoring.DoorOpen;
   "OtherSafetyInterface".InspectionExternalDoor.monitoring.DoorUnLock := "OtherSafetyInterface".InspectionExternalDoor.monitoring.DoorOpen;
   "OtherSafetyInterface".InspectionExternalDoor.monitoring.DoorClose := "SafetyDoorInterface".fDoor6Interface.monitoring.DoorClose AND "SafetyDoorInterface".fDoor7Interface.monitoring.DoorClose AND "SafetyDoorInterface".fDoor8Interface.monitoring.DoorClose;
   "OtherSafetyInterface".InspectionExternalDoor.monitoring.DoorLock := "OtherSafetyInterface".InspectionExternalDoor.monitoring.DoorClose;
END_REGION

REGION Network 29: Inspection BA030 Main Door
   RUNG wire#powerrail
      Contact( "SafetyDoorInterface".fDoor11Interface.monitoring.DoorOpen )
      wire#w1
      Coil( "OtherSafetyInterface".Inspection30MaintDoor.monitoring.DoorOpen )
   END_RUNG
   RUNG wire#w1
      Coil( "OtherSafetyInterface".Inspection30MaintDoor.monitoring.DoorUnLock )
   END_RUNG
   RUNG wire#powerrail
      Contact( "SafetyDoorInterface".fDoor11Interface.monitoring.DoorClose )
      wire#w2
      Coil( "OtherSafetyInterface".Inspection30MaintDoor.monitoring.DoorClose )
   END_RUNG
   RUNG wire#w2
      Coil( "OtherSafetyInterface".Inspection30MaintDoor.monitoring.DoorLock )
   END_RUNG
   // the same network as SCL:
   "OtherSafetyInterface".Inspection30MaintDoor.monitoring.DoorOpen := "SafetyDoorInterface".fDoor11Interface.monitoring.DoorOpen;
   "OtherSafetyInterface".Inspection30MaintDoor.monitoring.DoorUnLock := "SafetyDoorInterface".fDoor11Interface.monitoring.DoorOpen;
   "OtherSafetyInterface".Inspection30MaintDoor.monitoring.DoorClose := "SafetyDoorInterface".fDoor11Interface.monitoring.DoorClose;
   "OtherSafetyInterface".Inspection30MaintDoor.monitoring.DoorLock := "SafetyDoorInterface".fDoor11Interface.monitoring.DoorClose;
END_REGION

REGION Network 30: Inspection BA040 Main Door
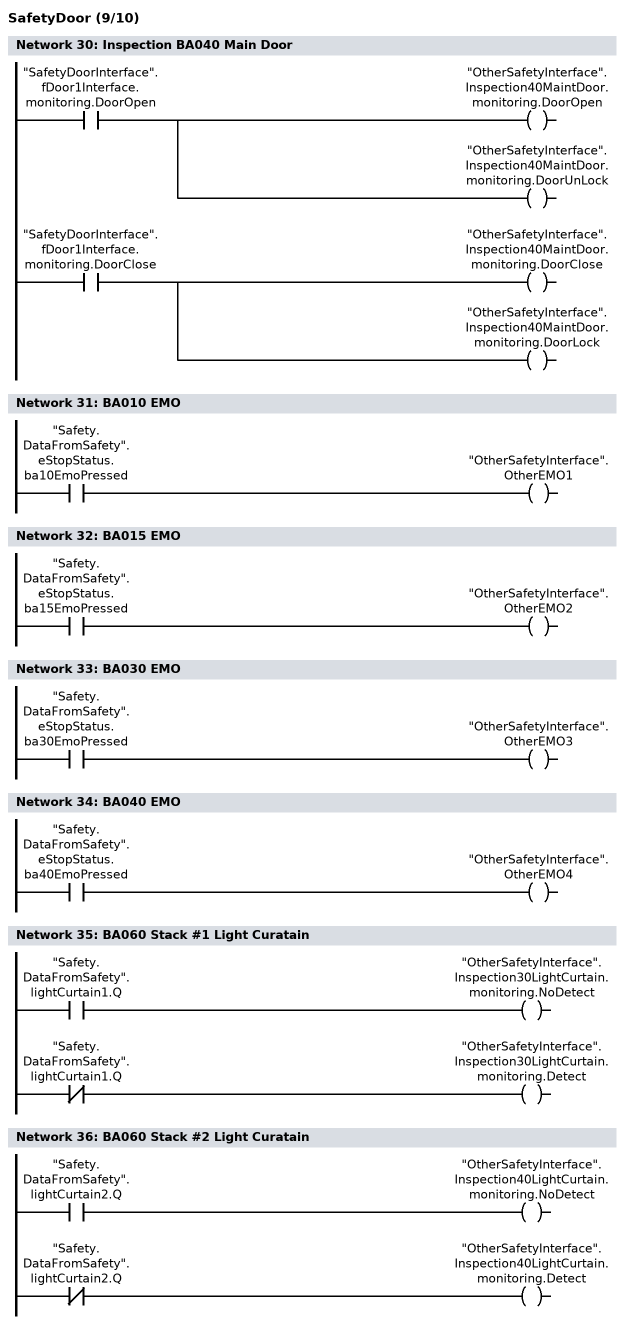
   RUNG wire#powerrail
      Contact( "SafetyDoorInterface".fDoor1Interface.monitoring.DoorOpen )
      wire#w1
      Coil( "OtherSafetyInterface".Inspection40MaintDoor.monitoring.DoorOpen )
   END_RUNG
   RUNG wire#w1
      Coil( "OtherSafetyInterface".Inspection40MaintDoor.monitoring.DoorUnLock )
   END_RUNG
   RUNG wire#powerrail
      Contact( "SafetyDoorInterface".fDoor1Interface.monitoring.DoorClose )
      wire#w2
      Coil( "OtherSafetyInterface".Inspection40MaintDoor.monitoring.DoorClose )
   END_RUNG
   RUNG wire#w2
      Coil( "OtherSafetyInterface".Inspection40MaintDoor.monitoring.DoorLock )
   END_RUNG
   // the same network as SCL:
   "OtherSafetyInterface".Inspection40MaintDoor.monitoring.DoorOpen := "SafetyDoorInterface".fDoor1Interface.monitoring.DoorOpen;
   "OtherSafetyInterface".Inspection40MaintDoor.monitoring.DoorUnLock := "SafetyDoorInterface".fDoor1Interface.monitoring.DoorOpen;
   "OtherSafetyInterface".Inspection40MaintDoor.monitoring.DoorClose := "SafetyDoorInterface".fDoor1Interface.monitoring.DoorClose;
   "OtherSafetyInterface".Inspection40MaintDoor.monitoring.DoorLock := "SafetyDoorInterface".fDoor1Interface.monitoring.DoorClose;
END_REGION

REGION Network 31: BA010 EMO
   RUNG wire#powerrail
      Contact( "Safety.DataFromSafety".eStopStatus.ba10EmoPressed )
      Coil( "OtherSafetyInterface".OtherEMO1 )
   END_RUNG
   // the same network as SCL:
   "OtherSafetyInterface".OtherEMO1 := "Safety.DataFromSafety".eStopStatus.ba10EmoPressed;
END_REGION

REGION Network 32: BA015 EMO
   RUNG wire#powerrail
      Contact( "Safety.DataFromSafety".eStopStatus.ba15EmoPressed )
      Coil( "OtherSafetyInterface".OtherEMO2 )
   END_RUNG
   // the same network as SCL:
   "OtherSafetyInterface".OtherEMO2 := "Safety.DataFromSafety".eStopStatus.ba15EmoPressed;
END_REGION

REGION Network 33: BA030 EMO
   RUNG wire#powerrail
      Contact( "Safety.DataFromSafety".eStopStatus.ba30EmoPressed )
      Coil( "OtherSafetyInterface".OtherEMO3 )
   END_RUNG
   // the same network as SCL:
   "OtherSafetyInterface".OtherEMO3 := "Safety.DataFromSafety".eStopStatus.ba30EmoPressed;
END_REGION

REGION Network 34: BA040 EMO
   RUNG wire#powerrail
      Contact( "Safety.DataFromSafety".eStopStatus.ba40EmoPressed )
      Coil( "OtherSafetyInterface".OtherEMO4 )
   END_RUNG
   // the same network as SCL:
   "OtherSafetyInterface".OtherEMO4 := "Safety.DataFromSafety".eStopStatus.ba40EmoPressed;
END_REGION

REGION Network 35: BA060 Stack #1 Light Curatain
   RUNG wire#powerrail
      Contact( "Safety.DataFromSafety".lightCurtain1.Q )
      Coil( "OtherSafetyInterface".Inspection30LightCurtain.monitoring.NoDetect )
   END_RUNG
   RUNG wire#powerrail
      I_Contact( "Safety.DataFromSafety".lightCurtain1.Q )
      Coil( "OtherSafetyInterface".Inspection30LightCurtain.monitoring.Detect )
   END_RUNG
   // the same network as SCL:
   "OtherSafetyInterface".Inspection30LightCurtain.monitoring.NoDetect := "Safety.DataFromSafety".lightCurtain1.Q;
   "OtherSafetyInterface".Inspection30LightCurtain.monitoring.Detect := NOT "Safety.DataFromSafety".lightCurtain1.Q;
END_REGION

REGION Network 36: BA060 Stack #2 Light Curatain
   RUNG wire#powerrail
      Contact( "Safety.DataFromSafety".lightCurtain2.Q )
      Coil( "OtherSafetyInterface".Inspection40LightCurtain.monitoring.NoDetect )
   END_RUNG
   RUNG wire#powerrail
      I_Contact( "Safety.DataFromSafety".lightCurtain2.Q )
      Coil( "OtherSafetyInterface".Inspection40LightCurtain.monitoring.Detect )
   END_RUNG
   // the same network as SCL:
   "OtherSafetyInterface".Inspection40LightCurtain.monitoring.NoDetect := "Safety.DataFromSafety".lightCurtain2.Q;
   "OtherSafetyInterface".Inspection40LightCurtain.monitoring.Detect := NOT "Safety.DataFromSafety".lightCurtain2.Q;
END_REGION

REGION Network 37: BA030 Cathode Conveyor Cover
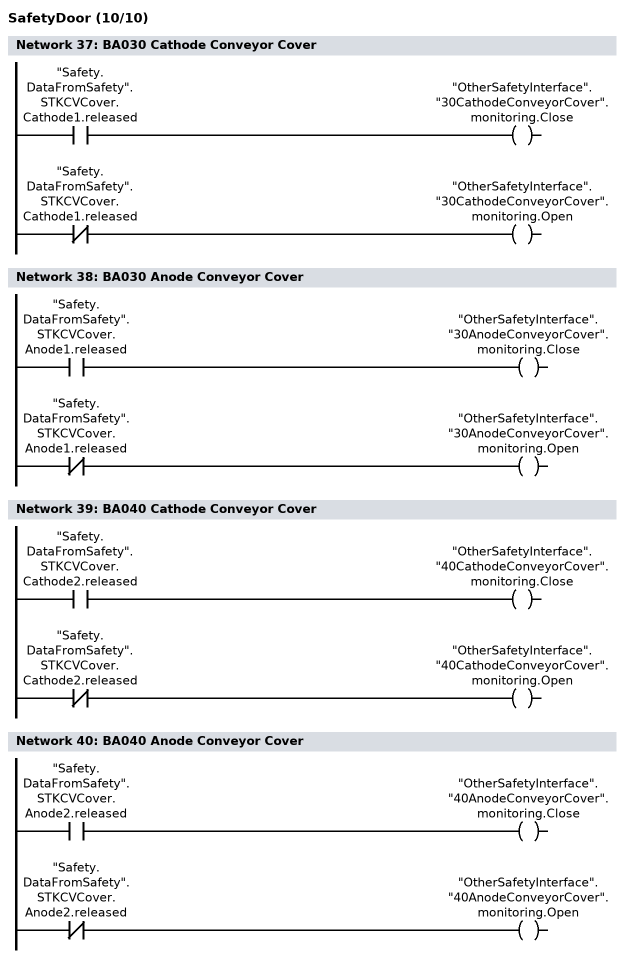
   RUNG wire#powerrail
      Contact( "Safety.DataFromSafety".STKCVCover.Cathode1.released )
      Coil( "OtherSafetyInterface"."30CathodeConveyorCover".monitoring.Close )
   END_RUNG
   RUNG wire#powerrail
      I_Contact( "Safety.DataFromSafety".STKCVCover.Cathode1.released )
      Coil( "OtherSafetyInterface"."30CathodeConveyorCover".monitoring.Open )
   END_RUNG
   // the same network as SCL:
   "OtherSafetyInterface"."30CathodeConveyorCover".monitoring.Close := "Safety.DataFromSafety".STKCVCover.Cathode1.released;
   "OtherSafetyInterface"."30CathodeConveyorCover".monitoring.Open := NOT "Safety.DataFromSafety".STKCVCover.Cathode1.released;
END_REGION

REGION Network 38: BA030 Anode Conveyor Cover
   RUNG wire#powerrail
      Contact( "Safety.DataFromSafety".STKCVCover.Anode1.released )
      Coil( "OtherSafetyInterface"."30AnodeConveyorCover".monitoring.Close )
   END_RUNG
   RUNG wire#powerrail
      I_Contact( "Safety.DataFromSafety".STKCVCover.Anode1.released )
      Coil( "OtherSafetyInterface"."30AnodeConveyorCover".monitoring.Open )
   END_RUNG
   // the same network as SCL:
   "OtherSafetyInterface"."30AnodeConveyorCover".monitoring.Close := "Safety.DataFromSafety".STKCVCover.Anode1.released;
   "OtherSafetyInterface"."30AnodeConveyorCover".monitoring.Open := NOT "Safety.DataFromSafety".STKCVCover.Anode1.released;
END_REGION

REGION Network 39: BA040 Cathode Conveyor Cover
   RUNG wire#powerrail
      Contact( "Safety.DataFromSafety".STKCVCover.Cathode2.released )
      Coil( "OtherSafetyInterface"."40CathodeConveyorCover".monitoring.Close )
   END_RUNG
   RUNG wire#powerrail
      I_Contact( "Safety.DataFromSafety".STKCVCover.Cathode2.released )
      Coil( "OtherSafetyInterface"."40CathodeConveyorCover".monitoring.Open )
   END_RUNG
   // the same network as SCL:
   "OtherSafetyInterface"."40CathodeConveyorCover".monitoring.Close := "Safety.DataFromSafety".STKCVCover.Cathode2.released;
   "OtherSafetyInterface"."40CathodeConveyorCover".monitoring.Open := NOT "Safety.DataFromSafety".STKCVCover.Cathode2.released;
END_REGION

REGION Network 40: BA040 Anode Conveyor Cover
   RUNG wire#powerrail
      Contact( "Safety.DataFromSafety".STKCVCover.Anode2.released )
      Coil( "OtherSafetyInterface"."40AnodeConveyorCover".monitoring.Close )
   END_RUNG
   RUNG wire#powerrail
      I_Contact( "Safety.DataFromSafety".STKCVCover.Anode2.released )
      Coil( "OtherSafetyInterface"."40AnodeConveyorCover".monitoring.Open )
   END_RUNG
   // the same network as SCL:
   "OtherSafetyInterface"."40AnodeConveyorCover".monitoring.Close := "Safety.DataFromSafety".STKCVCover.Anode2.released;
   "OtherSafetyInterface"."40AnodeConveyorCover".monitoring.Open := NOT "Safety.DataFromSafety".STKCVCover.Anode2.released;
END_REGION
END_FUNCTION

FUNCTION "IF_Bool_Mapping" : Void
{ S7_Optimized_Access := 'TRUE' ; Published := 'TRUE' }
VERSION : 0.1

BEGIN
	//Des : I/O Interface signal Mapping //
	
	REGION BK
	    
	    REGION BK01
	        "BK01"."X10-1 JR OUT P&P1 Y-AXIS ROBOT LIMIT SENSOR(-)" := "Sensor"."OUT P&P GRIPPER 1ST Y-AXIS LIMIT SENSOR(-)";
	        "BK01"."X11-1 JR OUT P&P1 Y-AXIS ROBOT LIMIT SENSOR(+)" := "Sensor"."OUT P&P GRIPPER 1ST Y-AXIS LIMIT SENSOR(+)";
	        "BK01"."X12-1 JR OUT P&P2 Y-AXIS ROBOT LIMIT SENSOR(-)" := "Sensor"."OUT P&P GRIPPER 2ND Y-AXIS LIMIT SENSOR(-)";
	        "BK01"."X13-1 JR OUT P&P2 Y-AXIS ROBOT LIMIT SENSOR(+)" := "Sensor"."OUT P&P GRIPPER 2ND Y-AXIS LIMIT SENSOR(+)";
	        "BK01"."X14-1 STACK 1 NG BOX DETECT SENSOR" := "BA060ZSIBK01.04";
	        "BK01"."X10-2 JR OUT P&P1 Y-AXIS ROBOT HOME SENSOR" := "Sensor"."OUT P&P GRIPPER 1ST Y-AXIS HOME SENSOR";
	        "BK01"."X12-2 JR OUT P&P2 Y-AXIS ROBOT HOME SENSOR" := "Sensor"."OUT P&P GRIPPER 2ND Y-AXIS HOME SENSOR";
	        "BK01"."X14-2 STACK 2 NG BOX DETECT SENSOR" := "BA060ZSIBK01.14";
	        
	    END_REGION;
	    REGION BK02
	        "BK02"."X10-1 JR OUT P&P1 Z-AXIS LIMIT SENSOR(-)" := "Sensor"."OUT P&P GRIPPER 1ST Z-AXIS LIMIT SENSOR(-)";
	        "BK02"."X10-2 JR OUT P&P1 Z-AXIS HOME SENSOR" := "Sensor"."OUT P&P GRIPPER 1ST Z-AXIS HOME SENSOR";
	        "BK02"."X12-1 JR OUT P&P1 Z-AXIS LIMIT SENSOR(+)" := "Sensor"."OUT P&P GRIPPER 1ST Z-AXIS LIMIT SENSOR(+)";
	        "BK02"."X12-2 JR OUT P&P1 STACK DETECT SENSOR" := "BA060ZSIBK02.03";
	        "BK02"."X14-1 JR OUT P&P1 CLAMP OPEN" := "BA060ZSIBK02.04";
	        "BK02"."X14-2 JR OUT P&P1 CLAMP CLOSE" := "BA060ZSIBK02.05";
	        "BK02"."X16-1 JR OUT P&P1 CLAMP OPEN/CLOSE PRESSURE SENSOR" := "BA060ZSIBK02.06";
	        "BK02"."X16-2 JR OUT P&P1 Z-AXIS SAFETY PIN LOADING SENSOR" := "BA060ZSIBK02.07";
	    END_REGION;
	    REGION BK03
	        "BK03"."X10-1 JR OUT P&P2 Z-AXIS LIMIT SENSOR(-)" := "Sensor"."OUT P&P GRIPPER 2ND Z-AXIS LIMIT SENSOR(-)";
	        "BK03"."X10-2 JR OUT P&P2 Z-AXIS HOME SENSOR" := "Sensor"."OUT P&P GRIPPER 2ND Z-AXIS HOME SENSOR";
	        "BK03"."X12-1 JR OUT P&P2 Z-AXIS LIMT SENSOR(+)" := "Sensor"."OUT P&P GRIPPER 2ND Z-AXIS LIMIT SENSOR(+)";
	        "BK03"."X12-2 JR OUT P&P2 STACK DETECT SENSOR" := "BA060ZSIBK03.03";
	        "BK03"."X14-1 JR OUT P&P2 CLAMP OPEN" := "BA060ZSIBK03.04";
	        "BK03"."X14-2 JR OUT P&P2 CLAMP CLOSE" := "BA060ZSIBK03.05";
	        "BK03"."X16-1 OUT P&P GRIPPER 2ND OPEN/CLOSE PRESSURE SENSOR" := "BA060ZSIBK03.06";
	        "BK03"."X16-2 OUT P&P GRIPPER 2ND Z-AXIS SAFETY PIN LOADING SENSOR" := "BA060ZSIBK03.07";
	    END_REGION ;
	    REGION BK04
	        "BK04"."X10-1 STACK #1 NG CLAMP MOVER OPEN" := "BA060ZSIBK04.00";
	        "BK04"."X11-1 STACK #1 NG CLAMP RIGHT OPEN" := "BA060ZSIBK04.01";
	        "BK04"."X12-1 STACK #1 NG CLAMP LEFT OPEN" := "BA060ZSIBK04.02";
	        "BK04"."X13-1 STAKC #1 NG CLAMP Z-AXIS UP" := "BA060ZSIBK04.03";
	        "BK04"."X14-1 STAKC #1 NG CLAMP MOVER BACKWARD" := "BA060ZSIBK04.04";
	        "BK04"."X15-1 STACK #1 NG BOX LIFT DOWN" := "BA060ZSIBK04.05";
	        "BK04"."X16-1 STACK #1 NG BOX LOCK DOWN" := "BA060ZSIBK04.06";
	        "BK04"."X17-1 STACK 1 NG BOX FULL SENSOR" := "BA060ZSIBK04.07";
	        "BK04"."X10-2 STACK #1 NG CLAMP MOVER CLOSE" := "BA060ZSIBK04.08";
	        "BK04"."X11-2 STACK #1 NG CLAMP RIGHT CLOSE" := "BA060ZSIBK04.09";
	        "BK04"."X12-2 STACK #1 NG CLAMP LEFT CLOSE" := "BA060ZSIBK04.10";
	        "BK04"."X13-2 STAKC #1 NG CLAMP Z-AXIS DOWN" := "BA060ZSIBK04.11";
	        "BK04"."X14-2 STAKC #1 NG CLAMP MOVER FORWARD" := "BA060ZSIBK04.12";
	        "BK04"."X15-2 STACK #1 NG BOX LIFT UP" := "BA060ZSIBK04.13";
	        "BK04"."X16-2 STACK #1 NG BOX LOCK UP" := "BA060ZSIBK04.14";
	    END_REGION ;
	    REGION BK05
	        "BK05"."X10-1 STACK #2 NG CLAMP MOVER OPEN" := "BA060ZSIBK05.00";
	        "BK05"."X11-1 STACK #2 NG CLAMP LEFT OPEN" := "BA060ZSIBK05.01";
	        "BK05"."X12-1 STACK #2 NG CLAMP RIGHT OPEN" := "BA060ZSIBK05.02";
	        "BK05"."X13-1 STAKC #2 NG CLAMP Z-AXIS UP" := "BA060ZSIBK05.03";
	        "BK05"."X14-1 STAKC #2 NG CLAMP MOVER BACKWARD" := "BA060ZSIBK05.04";
	        "BK05"."X15-1 STACK #2 NG BOX LIFT DOWN" := "BA060ZSIBK05.05";
	        "BK05"."X16-1 STACK #2 NG BOX LOCK DOWN" := "BA060ZSIBK05.06";
	        "BK05"."X17-1 STACK # NG BOX FULL SENSOR" := "BA060ZSIBK05.07";
	        "BK05"."X10-2 STACK #2 NG BOX LIFT DOWN" := "BA060ZSIBK05.08";
	        "BK05"."X11-2 STACK #2 NG CLAMP LEFT CLOSE" := "BA060ZSIBK05.09";
	        "BK05"."X12-2 STACK #2 NG CLAMP RIGHT CLOSE" := "BA060ZSIBK05.10";
	        "BK05"."X13-2 STAKC #2 NG CLAMP Z-AXIS DOWN" := "BA060ZSIBK05.11";
	        "BK05"."X14-2 STAKC #2 NG CLAMP MOVER FORWARD" := "BA060ZSIBK05.12";
	        "BK05"."X15-2 STACK #2 NG BOX LIFT UP" := "BA060ZSIBK05.13";
	        "BK05"."X16-2 STACK #2 NG BOX LOCK UP" := "BA060ZSIBK05.14";
	        
	    END_REGION ;
	    REGION BK06
	        "BK06"."X10-1 TOP TAPE DIAMETER SENSOR" := "BA060ZSIBK06.00";
	        "BK06"."X11-1 TOP TAPE CUTTER UP" := "BA060ZSIBK06.01";
	        "BK06"."X12-1 TOP TAPE CUTTER CLAMP UP" := "BA060ZSIBK06.02";
	        "BK06"."X13-1 TOP TAPE CLAMP OPEN" := "BA060ZSIBK06.03";
	        "BK06"."X14-1 TOP TAPE TENSION BACKWARD" := "BA060ZSIBK06.04";
	        "BK06"."X15-1 TOP TAPE LOADING BACKWARD" := "BA060ZSIBK06.05";
	        "BK06"."X11-2 TOP TAPE CUTTER DOWN" := "BA060ZSIBK06.09";
	        "BK06"."X12-2 TOP TAPE CUTTER CLAMP DOWN" := "BA060ZSIBK06.10";
	        "BK06"."X13-2 TOP TAPE CLAMP CLOSE" := "BA060ZSIBK06.11";
	        "BK06"."X14-2 TOP TAPE TENSION FORWARD" := "BA060ZSIBK06.12";
	        "BK06"."X15-2 TOP TAPE LOADING FORWARD" := "BA060ZSIBK06.13";
	        
	    END_REGION ;
	    REGION BK07
	        "BK07"."X10-1 TAPE ATTACHMENT VACUUM PRESSURE SWITCH" := "BA060ZSIBK07.00";
	        "BK07"."X12-1 TOP TAPE ATTACHMENT UP" := "BA060ZSIBK07.02";
	        "BK07"."X12-2 TOP TAPE ATTACHMENT DOWN" := "BA060ZSIBK07.03";
	        "BK07"."X14-1 TOP TAPING X-AXIS LIMIT SENSOR(-)" := "Sensor"."TAPE  Attachment ROBOT LIMIT SENSOR(-)";
	        "BK07"."X14-2 TOP TAPING X-AXIS HOMING SENSOR" := "Sensor"."TAPE  Attachment ROBOT HOMING SENSOR";
	        "BK07"."X16-1 TOP TAPING X-AXIS LIMIT SENSOR(+)" := "Sensor"."TAPE  Attachment ROBOT LIMIT SENSOR(+)";
	        
	        
	    END_REGION ;
	    REGION BK08
	        "BK08"."X10-1 TOP TAPE CLAMP TOP LEFT UP" := "BA060ZSIBK08.00";
	        "BK08"."X11-1 TOP TAPE CLAMP TOP CENTER UP" := "BA060ZSIBK08.01";
	        "BK08"."X12-1 TOP TAPE CLAMP TOP RIGHT UP" := "BA060ZSIBK08.02";
	        "BK08"."X13-1 TOP TAPE ATTACHMENT VACUUM PRESSURE SWITCH" := "BA060ZSIBK08.03";
	        "BK08"."X14-1 TOP TAPE CLAMP BTM DOWN" := "BA060ZSIBK08.04";
	        "BK08"."X15-1 TOP TAPING Y-AXIS LIMIT SENSOR(-)" := "Sensor"."TOP TAPE fix STAGE ROBOT LIMIT SENSOR(-)";
	        "BK08"."X16-1 TOP TAPING Y-AXIS LIMIT SENSOR(+)" := "Sensor"."TOP TAPE fix STAGE ROBOT LIMIT SENSOR(+)";
	        "BK08"."X17-1 TOP TAPE FIX STAGE STACK DETECT SENSOR" := "BA060ZSIBK08.07";
	        "BK08"."X10-2 TOP TAPE CLAMP TOP LEFT DOWN" := "BA060ZSIBK08.08";
	        "BK08"."X11-2 TOP TAPE CLAMP TOP CENTER DOWN" := "BA060ZSIBK08.09";
	        "BK08"."X12-2 TOP TAPE CLAMP TOP RIGHT DOWN" := "BA060ZSIBK08.10";
	        "BK08"."X14-2 TOP TAPE CLAMP BTM UP" := "BA060ZSIBK08.12";
	        "BK08"."X15-2 TOP TAPING Y-AXIS HOME SENSOR" := "Sensor"."TOP TAPE fix STAGE ROBOT HOME SENSOR";
	        
	        
	    END_REGION ;
	    REGION BK09
	        "BK09"."X10-1 SIDE TAPE CUTTER BACKWARD" := "BA060ZSIBK09.00";
	        "BK09"."X11-1 SIDE TAPE CUTTER CLAMP BACKWARD" := "BA060ZSIBK09.01";
	        "BK09"."X12-1 SIDE TAPE CLAMP OPEN" := "BA060ZSIBK09.02";
	        "BK09"."X13-1 SIDE TAPE TENSION BACKWARD" := "BA060ZSIBK09.03";
	        "BK09"."X14-1 SIDE TAPE LOADING BACKWARD" := "BA060ZSIBK09.04";
	        "BK09"."X15-1 SIDE TAPE DIAMETER SENSOR" := "BA060ZSIBK09.05";
	        "BK09"."X10-2 SIDE TAPE CUTTER FORWARD" := "BA060ZSIBK09.08";
	        "BK09"."X11-2 SIDE TAPE CUTTER CLAMP FORWARD" := "BA060ZSIBK09.09";
	        "BK09"."X12-2 SIDE TAPE CLAMP CLOSE" := "BA060ZSIBK09.10";
	        "BK09"."X13-2 SIDE TAPE TENSION FORWARD" := "BA060ZSIBK09.11";
	        "BK09"."X14-2 SIDE TAPE LOADING FORWARD" := "BA060ZSIBK09.12";
	        
	    END_REGION ;
	    REGION BK10
	        "BK10"."X10-1 SIDE TAPE Attachment LEFT BACKWARD" := "BA060ZSIBK10.00";
	        "BK10"."X11-1 SIDE TAPE Attachment RIGHT BACKWARD" := "BA060ZSIBK10.01";
	        "BK10"."X12-1 SIDE TAPE Attachment 1 TOP VACCUM PRESSURE SWITCH" := "BA060ZSIBK10.02";
	        "BK10"."X13-1 SIDE TAPE Attachment 2 TOP VACCUM PRESSURE SWITCH" := "BA060ZSIBK10.03";
	        "BK10"."X14-1 SIDE TAPE ATTACHEMNT LEFT PRESSURE SWITCH" := "BA060ZSIBK10.04";
	        "BK10"."X15-1 SIDE TAPE Attachment BTM BACKWARD" := "BA060ZSIBK10.05";
	        "BK10"."X16-1 SIDE TAPING Y-AYIS LIMIT SENSOR(-)" := "Sensor"."SIDE TAPE Attachment FORWARD/BACKWARD ROBOT LIMIT SENSOR(-)";
	        "BK10"."X17-1 SIDE TAPING Y-AYIS LIMIT SENSOR(+)" := "Sensor"."SIDE TAPE Attachment FORWARD/BACKWARD ROBOT LIMIT SENSOR(+)";
	        "BK10"."X10-2 SIDE TAPE Attachment LEFT FORWARD" := "BA060ZSIBK10.08";
	        "BK10"."X11-2 SIDE TAPE Attachment RIGHT FORWARD" := "BA060ZSIBK10.09";
	        "BK10"."X12-2 SIDE TAPE Attachment 1 BTM VACCUM PRESSURE SWITCH" := "BA060ZSIBK10.10";
	        "BK10"."X13-2 SIDE TAPE Attachment 2 BTM VACCUM PRESSURE SWITCH" := "BA060ZSIBK10.11";
	        "BK10"."X14-2 SIDE TAPE ATTACHMENT RIGHT PRESSURE SWITCH" := "BA060ZSIBK10.12";
	        "BK10"."X15-2 SIDE TAPE Attachment BTM FORWARD" := "BA060ZSIBK10.13";
	        "BK10"."X16-2 SIDE TAPING Y-AYIS HOME SENSOR" := "Sensor"."SIDE TAPE Attachment FORWARD/BACKWARD ROBOT HOME SENSOR";
	        
	    END_REGION ;
	    REGION BK11
	        "BK11"."X10-1 SIDE TAPING X-AXIS LIMIT SENSOR(-)" := "Sensor"."SIDE TAPE Attachment MOVER ROBOT LIMIT SENSOR(-)";
	        "BK11"."X11-1 SIDE TAPING X-AXIS LIMIT SENSOR(+)" := "Sensor"."SIDE TAPE Attachment MOVER ROBOT LIMIT SENSOR(+)";
	        "BK11"."X12-1 JR FIX STAGE X-AXIS LIMIT SENSOR(-)" := "Sensor"."SIDE TAPE fix Stage LIMIT SENSOR(-)";
	        "BK11"."X13-1 JR FIX STAGE X-AXIS LIMIT SENSOR(+)" := "Sensor"."SIDE TAPE fix Stage LIMIT SENSOR(+)";
	        "BK11"."X14-1 JR FIX STAGE C-AXIS LIMIT SENSOR(-)" := "Sensor"."SIDE TAPE fix Stage Rotation LIMIT SENSOR(-)";
	        "BK11"."X15-1 JR FIX STAGE C-AXIS LIMIT SENSOR(+)" := "Sensor"."SIDE TAPE fix Stage Rotation LIMIT SENSOR(+)";
	        "BK11"."X16-1 STACK DETECT SENSOR" := "BA060ZSIBK11.06";
	        "BK11"."X17-1 SIDE TAPE FIX STAGE OPEN" := "BA060ZSIBK11.07";
	        "BK11"."X10-2 SIDE TAPING X-AXIS HOME SENSOR" := "Sensor"."SIDE TAPE Attachment MOVER ROBOT HOME SENSOR";
	        "BK11"."X12-2 JR FIX STAGE X-AXIS HOMING SENSOR" := "Sensor"."SIDE TAPE FIX STAGE HOMING SENSOR";
	        "BK11"."X14-2 JR FIX STAGE X-AXIS HOMING SENSOR" := "Sensor"."SIDE TAPE FIX STAGE ROTATION HOMING SENSOR";
	        "BK11"."X16-2 SIDE TAPE CLAMP SAFETY PIN LOADING SENSOR" := "BA060ZSIBK11.14";
	        "BK11"."X17-2 SIDE TAPE FIX STAGE CLOSE" := "BA060ZSIBK11.15";
	        
	    END_REGION ;
	    REGION BK12
	        "BK12"."X10-1 SPARE" := "BA060ZSIBK12.00";
	        "BK12"."X11-1 SPARE" := "BA060ZSIBK12.01";
	        "BK12"."X12-1 HP STAGE LIFT #1 FRONT DOWN" := "BA060ZSIBK12.02";
	        "BK12"."X13-1 HP STAGE LIFT #1 REAR DOWN" := "BA060ZSIBK12.03";
	        "BK12"."X14-1 HP STACK DETECT SENSOR 1" := "BA060ZSIBK12.04";
	        "BK12"."X15-1 HP STAGE 1 SAFETY PIN LOADING SENSOR" := "BA060ZSIBK12.05";
	        "BK12"."X10-2 SPARE" := "BA060ZSIBK12.08";
	        "BK12"."X11-2 SPARE" := "BA060ZSIBK12.09";
	        "BK12"."X12-2 HP STAGE LIFT #1 FRONT UP" := "BA060ZSIBK12.10";
	        "BK12"."X13-2 HP STAGE LIFT #1 REAR UP" := "BA060ZSIBK12.11";
	        
	    END_REGION ;
	    REGION BK13
	        "BK13"."X10-1 SPARE" := "BA060ZSIBK13.00";
	        "BK13"."X11-1 SPARE" := "BA060ZSIBK13.01";
	        "BK13"."X12-1 HP STAGE LIFT #2 FRONT DOWN" := "BA060ZSIBK13.02";
	        "BK13"."X13-1 HP STAGE LIFT #2 REAR DOWN" := "BA060ZSIBK13.03";
	        "BK13"."X14-1 HP STACK DETECT SENSOR 2" := "BA060ZSIBK13.04";
	        "BK13"."X15-1 HP STAGE 2 SAFETY PIN LOADING SENSOR" := "BA060ZSIBK13.05";
	        "BK13"."X10-2 SPARE" := "BA060ZSIBK13.08";
	        "BK13"."X11-2 SPARE" := "BA060ZSIBK13.09";
	        "BK13"."X12-2 HP STAGE LIFT #2 FRONT UP" := "BA060ZSIBK13.10";
	        "BK13"."X13-2 HP STAGE LIFT #2 REAR UP" := "BA060ZSIBK13.11";
	        
	    END_REGION ;
	    REGION BK14
	        "BK14"."X10-1 HIPOT TAB CONTACTOR BACKWARD" := "BA060ZSIBK14.00";
	        "BK14"."X11-1 HIPOT TAB CONTACTOR LEFT OPEN" := "BA060ZSIBK14.01";
	        "BK14"."X12-1 HIPOT TAB CONTACTOR RIGHT OPEN" := "BA060ZSIBK14.02";
	        "BK14"."X13-1 SPARE" := "BA060ZSIBK14.03";
	        "BK14"."X14-1 SPARE" := "BA060ZSIBK14.04";
	        "BK14"."X15-1 HIPOT&THICKNESS STAGE LIFT FRONT DOWN" := "BA060ZSIBK14.05";
	        "BK14"."X16-1 HIPOT&THICKNESS STAGE LIFT REAR DOWN" := "BA060ZSIBK14.06";
	        "BK14"."X10-2 HIPOT TAB CONTACTOR FORWARD" := "BA060ZSIBK14.08";
	        "BK14"."X11-2 HIPOT TAB CONTACTOR LEFT CLOSE" := "BA060ZSIBK14.09";
	        "BK14"."X12-2 HIPOT TAB CONTACTOR RIGHT CLOSE" := "BA060ZSIBK14.10";
	        "BK14"."X13-2 SPARE" := "BA060ZSIBK14.11";
	        "BK14"."X14-2 SPARE" := "BA060ZSIBK14.12";
	        "BK14"."X15-2 INSPECTION STAGE LIFT FRONT UP" := "BA060ZSIBK14.13";
	        "BK14"."X16-2 INSPECTION STAGE LIFT REAR UP" := "BA060ZSIBK14.14";
	        
	    END_REGION ;
	    REGION BK15
	        "BK15"."X10-1 HIPOT&THICKNESS Z-AXIS LIMIT SENSOR(-)" := "Sensor"."Thickness Z-AXIS LIMIT SENSOR(-)";
	        "BK15"."X11-1 HIPOT&THICKNESS Z-AXIS LIMIT SENSOR(+)" := "Sensor"."Thickness Z-AXIS LIMIT SENSOR(+)";
	        "BK15"."X12-1 HIPOT&THICKNESS STACK DETECT SENSOR" := "BA060ZSIBK15.02";
	        "BK15"."X13-1 HI-POT SAFETY PIN LOADING SENSOR" := "BA060ZSIBK15.03";
	        "BK15"."X10-2 HIPOT&THICKNESS Z-AXIS HOME SENSOR" := "Sensor"."Thickness Z-AXIS HOME SENSOR";
	    END_REGION ;
	    REGION BK16
	        "BK16"."X10-1 FINAL VISION STAGE LIFT UP" := "BA060ZSIBK16.00";
	        "BK16"."X10-2 FINAL VISION STAGE LIFT DOWN" := "BA060ZSIBK16.01";
	        "BK16"."X12-1 FINAL VISION LIGHT UP" := "BA060ZSIBK16.02";
	        "BK16"."X12-2 FINAL VISION LIGHT DOWN" := "BA060ZSIBK16.03";
	        "BK16"."X14-1 FINAL VISION STAGE DETECT SENSOR" := "BA060ZSIBK16.04";
	        
	    END_REGION ;
	    REGION BK17
	        "BK17"."X10-1 LASER MARKING COVER UP" := "BA060ZSIBK17.00";
	        "BK17"."X10-2 LASER MARKING COVER DOWN" := "BA060ZSIBK17.01";
	        "BK17"."X12-1 LASER MARKING Stage Lift UP" := "BA060ZSIBK17.02";
	        "BK17"."X12-2 LASER MARKING Stage Lift DOWN" := "BA060ZSIBK17.03";
	        "BK17"."X14-2 LASER MARKING STACK DETECT SENSOR" := "BA060ZSIBK17.05";
	        "BK17"."X16-1 SPARE" := "BA060ZSIBK17.06";
	    END_REGION ;
	    REGION BK18
	        "BK18"."X10-1 WEIGHT NG CLAMP MOVER OPEN" := "BA060ZSIBK18.00";
	        "BK18"."X11-1 WEIGHT NG CLAMP LEFT OPEN" := "BA060ZSIBK18.01";
	        "BK18"."X12-1 WEIGHT NG CLAMP RIGHT OPEN" := "BA060ZSIBK18.02";
	        "BK18"."X13-1 WEIGHT NG CLAMP Z-AXIS UP" := "BA060ZSIBK18.03";
	        "BK18"."X14-1 WEIGHT NG CLAMP MOVER BACKWARD" := "BA060ZSIBK18.04";
	        "BK18"."X15-1 WEIGHT NG BOX LIFT DOWN" := "BA060ZSIBK18.05";
	        "BK18"."X16-1 WEIGHT NG BOX LOCK DOWN" := "BA060ZSIBK18.06";
	        "BK18"."X17-1 STACK NG FULL SENSOR" := "BA060ZSIBK18.07";
	        "BK18"."X10-2 WEIGHT NG CLAMP MOVER CLOSE" := "BA060ZSIBK18.08";
	        "BK18"."X11-2 WEIGHT NG CLAMP LEFT CLOSE" := "BA060ZSIBK18.09";
	        "BK18"."X12-2 WEIGHT NG CLAMP RIGHT CLOSE" := "BA060ZSIBK18.10";
	        "BK18"."X13-2 WEIGHT NG CLAMP Z-AXIS DOWN" := "BA060ZSIBK18.11";
	        "BK18"."X14-2 WEIGHT NG CLAMP MOVER FORWARD" := "BA060ZSIBK18.12";
	        "BK18"."X15-2 WEIGHT NG BOX LIFT UP" := "BA060ZSIBK18.13";
	        "BK18"."X16-2 WEIGHT NG BOX LOCK UP" := "BA060ZSIBK18.14";
	        "BK18"."X17-2 SPARE" := "BA060ZSIBK18.15";
	        
	    END_REGION ;
	    REGION BK19
	        "BK19"."X10-1 SPARE" := "BA060ZSIBK19.00";
	        "BK19"."X10-2 SPARE" := "BA060ZSIBK19.01";
	        "BK19"."X12-1 SPARE" := "BA060ZSIBK19.02";
	        "BK19"."X12-2 SPARE" := "BA060ZSIBK19.03";
	        "BK19"."X14-1 WEIGHT DETECT SENSOR" := "BA060ZSIBK19.04";
	        "BK19"."X16-1 MAIN VALVE DIGITAL PRESSURE SWITCH OUT1" := "BA060ZSIBK19.06";
	    END_REGION ;
	    REGION BK20
	        "BK20"."X10-1 INS TRANSFER P&P1 X-AXIS LIMIT SENSOR(-)" := "Sensor"."Process P&P X-axis Head#1 LIMIT SENSOR(-)";
	        "BK20"."X11-1 INS TRANSFER P&P1 X-AXIS LIMIT SENSOR(+)" := "Sensor"."Process P&P X-axis Head#1 LIMIT SENSOR(+)";
	        "BK20"."X12-1 INS TRANSFER P&P2 X-AXIS LIMIT SENSOR(-)" := "Sensor"."Process P&P X-axis Head#2 LIMIT SENSOR(-)";
	        "BK20"."X13-1 INS TRANSFER P&P2 X-AXIS LIMIT SENSOR(+)" := "Sensor"."Process P&P X-axis Head#2 LIMIT SENSOR(+)";
	        "BK20"."X10-2 INS TRANSFER P&P1 X-AXIS HOMING SENSOR" := "Sensor"."Process P&P X-axis Head#1 HOMING SENSOR";
	        "BK20"."X12-2 INS TRANSFER P&P2 X-AXIS HOMING SENSOR" := "Sensor"."Process P&P X-axis Head#2 HOMING SENSOR";
	        
	    END_REGION ;
	    REGION BK21
	        "BK21"."X10-1 INS TRANSFER P&P1 Y-AXIS LIMIT SENSOR(-)" := "Sensor"."Process P&P Y-axis Head#1 LIMIT SENSOR(-)";
	        "BK21"."X11-1 INS TRANSFER P&P1 Y-AXIS LIMIT SENSOR(+)" := "Sensor"."Process P&P Y-axis Head#1 LIMIT SENSOR(+)";
	        "BK21"."X12-1 INS TRANSFER P&P1 Z-AXIS LIMIT SENSOR(-)" := "Sensor"."Process P&P Z-axis Head#1 LIMIT SENSOR(-)";
	        "BK21"."X13-1 INS TRANSFER P&P1 Z-AXIS LIMIT SENSOR(+)" := "Sensor"."Process P&P Z-axis Head#1 LIMIT SENSOR(+)";
	        "BK21"."X14-1 INS TRANSFER P&P1 CLAMP OPEN SENSOR" := "BA060ZSIBK21.04";
	        "BK21"."X15-1 INS TRANSFER P&P1 CLAMP STACK DETECT SENSOR" := "BA060ZSIBK21.05";
	        "BK21"."X16-1 INS TRANSFER P&P1 Z-AXIS SAFETY PIN LOADING SENSOR" := "BA060ZSIBK21.06";
	        "BK21"."X10-2 INS TRANSFER P&P1 Y-AXIS HOMING SENSOR" := "Sensor"."Process P&P Y-axis Head#1 HOMING SENSOR";
	        "BK21"."X12-2 INS TRANSFER P&P1 Z-AXIS HOMING SENSOR" := "Sensor"."Process P&P Z-axis Head#1 HOMING SENSOR";
	        "BK21"."X14-2 INS TRANSFER P&P1 CLAMP CLOSE SENSOR" := "BA060ZSIBK21.12";
	        "BK21"."X15-2 INS TRANSFER P&P1 CLAMP OPEN/CLOSE PRESSURE SENSOR" := "BA060ZSIBK21.13";
	        
	    END_REGION ;
	    REGION BK22
	        "BK22"."X10-1 INS TRANSFER P&P2 Y-AXIS LIMIT SENSOR(-)" := "Sensor"."Process P&P Y-axis Head#2 LIMIT SENSOR(-)";
	        "BK22"."X11-1 INS TRANSFER P&P2 Y-AXIS LIMIT SENSOR(+)" := "Sensor"."Process P&P Y-axis Head#2 LIMIT SENSOR(+)";
	        "BK22"."X12-1 INS TRANSFER P&P2 Z-AXIS LIMIT SENSOR(-)" := "Sensor"."Process P&P Z-axis Head#2 LIMIT SENSOR(-)";
	        "BK22"."X13-1 INS TRANSFER P&P2 Z-AXIS LIMIT SENSOR(+)" := "Sensor"."Process P&P Z-axis Head#2 LIMIT SENSOR(+)";
	        "BK22"."X14-1 INS TRANSFER P&P2 CLAMP OPEN SENSOR" := "BA060ZSIBK22.04";
	        "BK22"."X15-1 INS TRANSFER P&P2 CLAMP STACK DETECT SENSOR" := "BA060ZSIBK22.05";
	        "BK22"."X16-1 INS TRANSFER P&P2 Z-AXIS SAFETY PIN LOADING SENSOR" := "BA060ZSIBK22.06";
	        "BK22"."X10-2 INS TRANSFER P&P2 Y-AXIS HOMING SENSOR" := "Sensor"."Process P&P Y-axis Head#2 HOMING SENSOR";
	        "BK22"."X12-2 PROCESS P&P Z-AXIS HEAD2 HOMING SENSOR" := "Sensor"."Process P&P Z-axis Head#2 HOMING SENSOR";
	        "BK22"."X14-2 INS TRANSFER P&P2 CLAMP CLOSE SENSOR" := "BA060ZSIBK22.12";
	        "BK22"."X15-2 INS TRANSFER P&P2 CLAMP OPEN/CLOSE PRESSURE SENSOR" := "BA060ZSIBK22.13";
	        
	    END_REGION ;
	    REGION BK23
	        "BK23"."X10-1 JR Unloading P&P Y-AXIS LIMIT SENSOR(-)" := "Sensor"."Unloading P&P X-axis LIMIT SENSOR(-)";
	        "BK23"."X11-1 JR Unloading P&P Y-AXIS LIMIT SENSOR(+)" := "Sensor"."Unloading P&P X-axis LIMIT SENSOR(+)";
	        "BK23"."X12-1 JR Unloading P&P Z-AXIS LIMIT SENSOR(-)" := "Sensor"."Unloading P&P Z-axis LIMIT SENSOR(-)";
	        "BK23"."X13-1 JR Unloading P&P Z-AXIS LIMIT SENSOR(+)" := "Sensor"."Unloading P&P Z-axis LIMIT SENSOR(+)";
	        "BK23"."X14-1 JR Unloading P&P C-AXIS LIMIT SENSOR(-)" := "Sensor"."Unloading P&P Θ-axis LIMIT SENSOR(-)";
	        "BK23"."X15-1 JR Unloading P&P C-AXIS LIMIT SENSOR(+)" := "Sensor"."Unloading P&P Θ-axis LIMIT SENSOR(+)";
	        "BK23"."X16-1 JR Unloading P&P CLAMP OPEN SENSOR" := "BA060ZSIBK23.06";
	        "BK23"."X17-1 JR Unloading P&P CLAMP STACK DETECT SENSOR" := "Sensor"."Unloading P&P X-axis HOMING SENSOR";
	        "BK23"."X10-2 JR Unloading P&P Y-AXIS HOMING SENSOR" := "Sensor"."Unloading P&P Z-axis HOMING SENSOR";
	        "BK23"."X12-2 JR Unloading P&P Z-AXIS HOMING SENSOR" := "Sensor"."Unloading P&P Z-axis HOMING SENSOR";
	        "BK23"."X14-2 JR Unloading P&P C-AXIS HOMING SENSOR" := "Sensor"."Unloading P&P Θ-axis HOMING SENSOR";
	        "BK23"."X16-2 JR Unloading P&P CLAMP CLOSE SENSOR" := "BA060ZSIBK23.14";
	        "BK23"."X17-2 JR Unloading P&P Z-AXIS SAFETY PIN LOADING SENSOR" := "BA060ZSIBK23.15";
	        
	    END_REGION ;
	    REGION BK24
	        "BK24"."X10-1 SIDE TAPE ATTACHMENT #1 TOP VACUUM ON" := "BA060ZSIBK24.00";
	        "BK24"."X10-2 SIDE TAPE ATTACHMENT #1 TOP VACUUM OFF" := "BA060ZSIBK24.01";
	        "BK24"."X12-1 SIDE TAPE ATTACHMENT #1 BTM VACUUM ON" := "BA060ZSIBK24.02";
	        "BK24"."X12-2 SIDE TAPE ATTACHMENT #1 BTM VACUUM OFF" := "BA060ZSIBK24.03";
	        "BK24"."X14-1 SIDE TAPE ATTACHMENT #2 TOP VACUUM ON" := "BA060ZSIBK24.04";
	        "BK24"."X14-2 SIDE TAPE ATTACHMENT #2 TOP VACUUM OFF" := "BA060ZSIBK24.05";
	        "BK24"."X16-1 SIDE TAPE ATTACHMENT #2 BTM VACUUM ON" := "BA060ZSIBK24.06";
	        "BK24"."X16-2 SIDE TAPE ATTACHMENT #2 BTM VACUUM OFF" := "BA060ZSIBK24.07";
	    END_REGION ;
	    REGION BK25
	        "BK25"."X10-1 TOP TAPE ATTACHMENT #1 VACUUM ON" := "BA060ZSIBK25.00";
	        "BK25"."X10-2 TOP TAPE ATTACHMENT #1 VACUUM OFF" := "BA060ZSIBK25.01";
	    END_REGION ;
	END_REGION
	REGION PM
	    REGION PM1
	        "PM1"."STACK #1 NG CLAMP MOVER CLOSE" := "BA060ZSIPM01.00";
	        "PM1"."STACK #1 NG CLAMP MOVER OPEN" := "BA060ZSIPM01.01";
	        "PM1"."STACK #1 NG CLAMP RIGHT CLOSE" := "BA060ZSIPM01.02";
	        "PM1"."STACK #1 NG CLAMP RIGHT OPEN" := "BA060ZSIPM01.03";
	        "PM1"."STACK #1 NG CLAMP LEFT OPEN" := "BA060ZSIPM01.04";
	        "PM1"."STACK #1 NG CLAMP LEFT CLOSE" := "BA060ZSIPM01.05";
	        "PM1"."STAKC #1 NG CLAMP Z-AXIS UP" := "BA060ZSIPM01.06";
	        "PM1"."STAKC #1 NG CLAMP Z-AXIS DOWN" := "BA060ZSIPM01.07";
	        "PM1"."STAKC #1 NG CLAMP MOVER FORWARD" := "BA060ZSIPM01.10";
	        "PM1"."STAKC #1 NG CLAMP MOVER BACKWARD" := "BA060ZSIPM01.11";
	        "PM1"."STACK #1 NG BOX LIFT UP" := "BA060ZSIPM01.12";
	        "PM1"."STACK #1 NG BOX LIFT DOWN" := "BA060ZSIPM01.13";
	        "PM1"."STACK #1 NG BOX LOCK UP" := "BA060ZSIPM01.14";
	        "PM1"."STACK #1 NG BOX LOCK DOWN" := "BA060ZSIPM01.15";
	        "PM1"."JR OUT P&P#1 CLAMP CLOSE" := "BA060ZSIPM01.16";
	        "PM1"."JR OUT P&P#1 CLAMP OPEN" := "BA060ZSIPM01.17";
	    END_REGION;
	    REGION PM2
	        "PM2"."STACK #2 NG CLAMP MOVER CLOSE" := "BA060ZSIPM02.00";
	        "PM2"."STACK #2 NG CLAMP MOVER OPEN" := "BA060ZSIPM02.01";
	        "PM2"."STACK #2 NG CLAMP LEFT CLOSE" := "BA060ZSIPM02.02";
	        "PM2"."STACK #2 NG CLAMP LEFT OPEN" := "BA060ZSIPM02.03";
	        "PM2"."STACK #2 NG CLAMP RIGHT CLOSE" := "BA060ZSIPM02.04";
	        "PM2"."STACK #2 NG CLAMP RIGHT OPEN" := "BA060ZSIPM02.05";
	        "PM2"."STAKC #2 NG CLAMP Z-AXIS UP" := "BA060ZSIPM02.06";
	        "PM2"."STAKC #2 NG CLAMP Z-AXIS DOWN" := "BA060ZSIPM02.07";
	        "PM2"."STAKC #2 NG CLAMP MOVER FORWARD" := "BA060ZSIPM02.10";
	        "PM2"."STAKC #2 NG CLAMP MOVER BACKWARD" := "BA060ZSIPM02.11";
	        "PM2"."STACK #2 NG BOX LIFT UP" := "BA060ZSIPM02.12";
	        "PM2"."STACK #2 NG BOX LIFT DOWN" := "BA060ZSIPM02.13";
	        "PM2"."STACK #2 NG BOX LOCK UP" := "BA060ZSIPM02.14";
	        "PM2"."STACK #2 NG BOX LOCK DOWN" := "BA060ZSIPM02.15";
	        "PM2"."JR OUT P&P#2 CLAMP CLOSE" := "BA060ZSIPM02.16";
	        "PM2"."JR OUT P&P#2 CLAMP OPEN" := "BA060ZSIPM02.17";
	    END_REGION;
	    REGION PM3
	        "PM3"."TOP TAPE CUTTER UP" := "BA060ZSIPM03.00";
	        "PM3"."TOP TAPE CUTTER DOWN" := "BA060ZSIPM03.01";
	        "PM3"."TOP TAPE CUTTER CLAMP UP" := "BA060ZSIPM03.02";
	        "PM3"."TOP TAPE CUTTER CLAMP DOWN" := "BA060ZSIPM03.03";
	        "PM3"."TOP TAPE CLAMP OPEN" := "BA060ZSIPM03.04";
	        "PM3"."TOP TAPE CLAMP CLOSE" := "BA060ZSIPM03.05";
	        "PM3"."TOP TAPE TENSION FORWARD" := "BA060ZSIPM03.06";
	        "PM3"."TOP TAPE TENSION BACKWARD" := "BA060ZSIPM03.07";
	        "PM3"."TOP TAPE LOADING FORWARD" := "BA060ZSIPM03.10";
	        "PM3"."TOP TAPE LOADING BACKWARD" := "BA060ZSIPM03.11";
	        "PM3"."TOP TAPE ATTACHMENT UP" := "BA060ZSIPM03.12";
	        "PM3"."TOP TAPE ATTACHMENT DOWN" := "BA060ZSIPM03.13";
	    END_REGION;
	    REGION PM4
	        "PM4"."TOP TAPE Clamp TOP LEFT UP" := "BA060ZSIPM04.00";
	        "PM4"."TOP TAPE Clamp TOP LEFT DOWN" := "BA060ZSIPM04.01";
	        "PM4"."TOP TAPE Clamp TOP CENTER UP" := "BA060ZSIPM04.02";
	        "PM4"."TOP TAPE Clamp TOP CENTER DOWN" := "BA060ZSIPM04.03";
	        "PM4"."TOP TAPE Clamp TOP RIGHT UP" := "BA060ZSIPM04.04";
	        "PM4"."TOP TAPE Clamp TOP RIGHT DOWN" := "BA060ZSIPM04.05";
	        "PM4"."TOP TAPE Clamp BTM UP" := "BA060ZSIPM04.06";
	        "PM4"."TOP TAPE Clamp BTM DOWN" := "BA060ZSIPM04.07";
	        
	    END_REGION;
	    REGION PM5
	        "PM5"."SIDE TAPE CUTTER FORWARD" := "BA060ZSIPM05.00";
	        "PM5"."SIDE TAPE CUTTER BACKWARD" := "BA060ZSIPM05.01";
	        "PM5"."SIDE TAPE CUTTER CLAMP FORWARD" := "BA060ZSIPM05.02";
	        "PM5"."SIDE TAPE CUTTER CLAMP BACKWARD" := "BA060ZSIPM05.03";
	        "PM5"."SIDE TAPE CLAMP CLOSE" := "BA060ZSIPM05.04";
	        "PM5"."SIDE TAPE CLAMP OPEN" := "BA060ZSIPM05.05";
	        "PM5"."SIDE TAPE TENSION FORWARD" := "BA060ZSIPM05.06";
	        "PM5"."SIDE TAPE TENSION BACKWARD" := "BA060ZSIPM05.07";
	        "PM5"."SIDE TAPE LOADING FORWARD" := "BA060ZSIPM05.10";
	        "PM5"."SIDE TAPE LOADING BACKWARD" := "BA060ZSIPM05.11";
	    END_REGION;
	    REGION PM6
	        
	        "PM6"."SIDE TAPE FIX STAGE CLOSE" := "BA060ZSIPM06.00";
	        "PM6"."SIDE TAPE FIX STAGE OPEN" := "BA060ZSIPM06.01";
	        "PM6"."SIDE TAPE Attachment LEFT FORWARD" := "BA060ZSIPM06.02";
	        "PM6"."SIDE TAPE Attachment LEFT BACKWARD" := "BA060ZSIPM06.03";
	        "PM6"."SIDE TAPE Attachment RIGHT FORWARD" := "BA060ZSIPM06.04";
	        "PM6"."SIDE TAPE Attachment RIGHT BACKWARD" := "BA060ZSIPM06.05";
	        "PM6"."SIDE TAPE Attachment BTM FORWARD" := "BA060ZSIPM06.06";
	        "PM6"."SIDE TAPE Attachment BTM BACKWARD" := "BA060ZSIPM06.07";
	    END_REGION;
	    REGION PM7
	        "PM7".SPARE := "BA060ZSIPM07.00";
	        "PM7".SPARE_1 := "BA060ZSIPM07.01";
	        "PM7".SPARE_2 := "BA060ZSIPM07.02";
	        "PM7".SPARE_3 := "BA060ZSIPM07.03";
	        "PM7".SPARE_4 := "BA060ZSIPM07.04";
	        "PM7".SPARE_5 := "BA060ZSIPM07.05";
	        "PM7".SPARE_6 := "BA060ZSIPM07.06";
	        "PM7".SPARE_7 := "BA060ZSIPM07.07";
	        "PM7"."HP STAGE LIFT #1 FRONT UP" := "BA060ZSIPM07.11";
	        "PM7"."HP STAGE LIFT #1 FRONT DOWN" := "BA060ZSIPM07.10";
	        "PM7"."HP STAGE LIFT #1 REAR UP" := "BA060ZSIPM07.13";
	        "PM7"."HP STAGE LIFT #1 REAR DOWN" := "BA060ZSIPM07.12";
	        "PM7"."HP STAGE LIFT #2 FRONT UP" := "BA060ZSIPM07.15";
	        "PM7"."HP STAGE LIFT #2 FRONT DOWN" := "BA060ZSIPM07.14";
	        "PM7"."HP STAGE LIFT #2 REAR UP" := "BA060ZSIPM07.17";
	        "PM7"."HP STAGE LIFT #2 REAR DOWN" := "BA060ZSIPM07.16";
	    END_REGION;
	    REGION PM8
	        "PM8"."HIPOT TAB CONTACTOR FORWARD" := "BA060ZSIPM08.00";
	        "PM8"."HIPOT TAB CONTACTOR BACKWARD" := "BA060ZSIPM08.01";
	        "PM8"."HIPOT TAB CONTACTOR LEFT CLOSE" := "BA060ZSIPM08.03";
	        "PM8"."HIPOT TAB CONTACTOR LEFT OPEN" := "BA060ZSIPM08.02";
	        "PM8"."HIPOT TAB CONTACTOR RIGHT CLOSE" := "BA060ZSIPM08.05";
	        "PM8"."HIPOT TAB CONTACTOR RIGHT OPEN" := "BA060ZSIPM08.04";
	        "PM8".SPARE := "BA060ZSIPM08.06";
	        "PM8".SPARE_1 := "BA060ZSIPM08.07";
	        "PM8".SPARE_2 := "BA060ZSIPM08.10";
	        "PM8".SPARE_3 := "BA060ZSIPM08.11";
	        "PM8"."HIPOT & THICKNESS STAGE LIFT FRONT UP" := "BA060ZSIPM08.12";
	        "PM8"."HIPOT & THICKNESS STAGE LIFT FRONT DOWN" := "BA060ZSIPM08.13";
	        "PM8"."HIPOT & THICKNESS STAGE LIFT REAR UP" := "BA060ZSIPM08.14";
	        "PM8"."HIPOT & THICKNESS STAGE LIFT REAR DOWN" := "BA060ZSIPM08.15";
	        
	        
	    END_REGION;
	    REGION PM9
	        "PM9"."FINAL VISION STAGE LIFT UP" := "BA060ZSIPM09.01";
	        "PM9"."FINAL VISION STAGE LIFT DOWN" := "BA060ZSIPM09.00";
	        "PM9"."FINAL VISION LIGHT UP" := "BA060ZSIPM09.03";
	        "PM9"."FINAL VISION LIGHT DOWN" := "BA060ZSIPM09.02";
	        "PM9"."LASER MARKING COVER UP" := "BA060ZSIPM09.05";
	        "PM9"."LASER MARKING COVER DOWN" := "BA060ZSIPM09.04";
	        "PM9"."LASER MARKING STAGE LIFT UP" := "BA060ZSIPM09.07";
	        "PM9"."LASER MARKING STAGE LIFT DOWN" := "BA060ZSIPM09.06";
	        "PM9".SPARE := "BA060ZSIPM09.11";
	        "PM9"."INS TRANSFER P&P CLAMP #1 CLOSE" := "BA060ZSIPM09.13";
	        "PM9"."INS TRANSFER P&P CLAMP #1 OPEN" := "BA060ZSIPM09.12";
	        "PM9"."INS TRANSFER P&P CLAMP #2 CLOSE" := "BA060ZSIPM09.15";
	        "PM9"."INS TRANSFER P&P CLAMP #2 OPEN" := "BA060ZSIPM09.14";
	        "PM9"."JR Unloading P&P CLAMP CLOSE" := "BA060ZSIPM09.17";
	        "PM9"."JR Unloading P&P CLAMP OPEN" := "BA060ZSIPM09.16";
	        
	    END_REGION;
	    REGION PM10
	        "PM10"."STACK NG CLAMP MOVER CLOSE" := "BA060ZSIPM10.01";
	        "PM10"."STACK NG CLAMP MOVER OPEN" := "BA060ZSIPM10.00";
	        "PM10"."STACK NG CLAMP LEFT CLOSE" := "BA060ZSIPM10.03";
	        "PM10"."STACK NG CLAMP LEFT OPEN" := "BA060ZSIPM10.02";
	        "PM10"."STACK NG CLAMP RIGHT CLOSE" := "BA060ZSIPM10.05";
	        "PM10"."STACK NG CLAMP RIGHT OPEN" := "BA060ZSIPM10.04";
	        "PM10"."STACK NG CLAMP Z-AXIS UP" := "BA060ZSIPM10.07";
	        "PM10"."STACK NG CLAMP Z-AXIS DOWN" := "BA060ZSIPM10.06";
	        "PM10"."STACK NG CLAMP MOVER FORWARD" := "BA060ZSIPM10.11";
	        "PM10"."STACK NG CLAMP MOVER BACKWARD" := "BA060ZSIPM10.10";
	        "PM10"."STACK NG BOX LIFT UP" := "BA060ZSIPM10.12";
	        "PM10"."STACK NG BOX LIFT DOWN" := "BA060ZSIPM10.13";
	        "PM10"."STACK NG BOX LOCK UP" := "BA060ZSIPM10.14";
	        "PM10"."STACK NG BOX LOCK DOWN" := "BA060ZSIPM10.15";
	        
	    END_REGION;
	END_REGION
	REGION SBK
	    REGION SBK1
	        "SBK1"."X1-1 EMO01 CH.A" := "BA060AZSISBK01.00";
	        "SBK1"."X2-1 EMO02 CH.A" := "BA060AZSISBK01.03";
	        "SBK1"."X3-1 EMO03 CH.A" := "BA060AZSISBK01.01";
	        "SBK1"."X4-1 EMO04 CH.A" := "BA060AZSISBK01.02";
	        
	        
	        
	        
	    END_REGION ;
	    REGION SBK2
	    END_REGION ;
	    REGION SBK3
	        "SBK3"."X1-1 GATE EC STACK 1 NG BOX PB.LOCK" := "BA060AZSISBK03.00";
	        "SBK3"."X2-1 GATE EC STACK 1 NG BOX PB.RESET" := "BA060AZSISBK03.01";
	        "SBK3"."X1-2 GATE EC STACK 1 NG BOX PB.UNLOCK" := "BA060AZSISBK03.04";
	        
	    END_REGION ;
	    REGION SBK4
	        "SBK4"."X1-1 GATE EC STACK 2 NG BOX PB.LOCK" := "BA060AZSISBK04.00";
	        "SBK4"."X2-1 GATE EC STACK 2 NG BOX PB.RESET" := "BA060AZSISBK04.01";
	        "SBK4"."X1-2 GATE EC STACK 2 NG BOX PB.UNLOCK" := "BA060AZSISBK04.04";
	    END_REGION ;
	    REGION SBK5
	        "SBK5"."X1-1 SCS BOX SCS MODE SLELECT SS.SETUP" := "BA060AZSISBK05.00";
	        "SBK5"."X2-1 SCS BOX SCS MODE SLELECT SS.DISABLE" := "BA060AZSISBK05.01";
	        "SBK5"."X1-2 SCS BOX SCS MODE SLELECT SS.AUTO" := "BA060AZSISBK05.04";
	        
	    END_REGION ;
	    REGION SBK6
	        "SBK6"."X1-1 GATE EC SIDE TAPE PB.LOCK" := "BA060AZSISBK06.00";
	        "SBK6"."X2-1 GATE EC SIDE TAPE PB.RESET" := "BA060AZSISBK06.01";
	        "SBK6"."X1-2 GATE EC SIDE TAPE PB.UNLOCK" := "BA060AZSISBK06.04";
	    END_REGION ;
	    REGION SBK7
	        "SBK7"."X1-1 GATE EC UNLOAD P&P PB.LOCK" := "BA060AZSISBK07.00";
	        "SBK7"."X2-1 GATE EC UNLOAD P&P PB.RESET" := "BA060AZSISBK07.01";
	        "SBK7"."X1-2 GATE EC UNLOAD P&P PB.UNLOCK" := "BA060AZSISBK07.04";
	    END_REGION ;
	    REGION SBK8
	    END_REGION ;
	    REGION SBK9
	        "SBK9"."X1-2 SAFETY DOOR LOCK1.INPUT" := "BA060AZSISBK09.00";
	        "SBK9"."X2-2 SAFETY DOOR LOCK2.INPUT" := "BA060AZSISBK09.01";
	        "SBK9"."X3-2 SAFETY DOOR LOCK3.INPUT" := "BA060AZSISBK09.02";
	    END_REGION ;
	    REGION SBK10
	        "SBK10"."X1-2 SAFETY DOOR LOCK4.INPUT" := "BA060AZSISBK10.00";
	        "SBK10"."X2-2 SAFETY DOOR LOCK5.INPUT" := "BA060AZSISBK10.01";
	        "SBK10"."X3-2 SAFETY DOOR LOCK6.INPUT" := "BA060AZSISBK10.02";
	    END_REGION ;
	    REGION SBK11
	        "SBK11"."X1-2 SAFETY DOOR LOCK7.INPUT" := "BA060AZSISBK11.00";
	        "SBK11"."X2-2 SAFETY DOOR LOCK8.INPUT" := "BA060AZSISBK11.01";
	        "SBK11"."X3-2 SAFETY DOOR LOCK9.INPUT" := "BA060AZSISBK11.02";
	    END_REGION ;
	    REGION SBK12
	        "SBK12"."X1-2 SAFETY DOOR LOCK10.INPUT" := "BA060AZSISBK12.00";
	        "SBK12"."X2-2 SAFETY DOOR LOCK11.INPUT" := "BA060AZSISBK12.01";
	        "SBK12"."X3-2 SAFETY DOOR LOCK12.INPUT" := "BA060AZSISBK12.02";
	    END_REGION ;
	    REGION SBK13
	        "SBK13"."X1-2 SAFETY DOOR LOCK13.INPUT" := "BA060AZSISBK13.00";
	    END_REGION ;
	END_REGION
	REGION MP
	    REGION MP101
	        "MP101"."KISTLER 100KN PRESS POWER TRIPPED E202CB" := "BA060AZSIMP101.00";
	        "MP101"."KISTLER 100KN PRESS POWER TRIPPED E208CB" := "BA060AZSIMP101.01";
	        "MP101"."KISTLER 30KN PRESS POWER TRIPPED E214CB" := "BA060AZSIMP101.02";
	        "MP101".SPARE := "BA060AZSIMP101.03";
	        
	        "MP101".SPARE_1 := "BA060AZSIMP101.04";
	        
	        "MP101"."E8404PWS CONTROLLER POWER SMPS AC POWER TRIPPED E320CB" := "BA060AZSIMP101.05";
	        "MP101"."E8704PWS SAFETY POWER SMPS AC POWER TRIPPED E326CB" := "BA060AZSIMP101.06";
	        "MP101"."E8804PWS CONTRL POWER SMPS AC POWER TRIPPED E332CB" := "BA060AZSIMP101.07";
	        "MP101"."PROCESSOR POWER ON TIPPRED E4120CB" := "BA060AZSIMP101.10";
	        
	        "MP101"."PROGRAMING POWER OUTLET TRPPED E4126CB" := "BA060AZSIMP101.11";
	        "MP101".SPARE_2 := "BA060AZSIMP101.12";
	        "MP101"."PANEL LED POWER TRIPPED E4304CB" := "BA060AZSIMP101.13";
	        "MP101".SPARE_3 := "BA060AZSIMP101.14";
	        "MP101"."PLC POWER SMPS DC OK E4404PWS" := "BA060AZSIMP101.15";
	        "MP101"."CONTROL LEVEL HUB POWER TRIPPED E4420CB" := "BA060AZSIMP101.16";
	        "MP101"."MAIN HMI POWER TRIPPED E4426CB" := "BA060AZSIMP101.17";
	        "MP101"."PORTABLE HMI POWER TIPPED E4432CB" := "BA060AZSIMP101.20";
	        "MP101"."PORTABLE HMI POWER TIPPED E4456CB" := "BA060AZSIMP101.21";
	        "MP101"."120VAC HEATER-1 POWER TR PRIMARY TRIPPED E5100CB" := "BA060AZSIMP101.22";
	        "MP101".SPARE_4 := "BA060AZSIMP101.23";
	        "MP101".SPARE_5 := "BA060AZSIMP101.24";
	        "MP101"."UPPER 1-1 HEATER POWER TRIPPED E5156CB" := "BA060AZSIMP101.25";
	        "MP101"."UPPER 1-2 HEATER POWER TRIPPED E5162CB" := "BA060AZSIMP101.26";
	        "MP101"."LOWER 1-1 HEATER POWER TRIPPED E5168CB" := "BA060AZSIMP101.27";
	        "MP101"."LOWER 1-2 HEATER POWER TRIPPED E5174CB" := "BA060AZSIMP101.30";
	        "MP101"."LOWER 1-3 HEATER POWER TRIPPED E5180CB" := "BA060AZSIMP101.31";
	        "MP101".SPARE_6 := "BA060AZSIMP101.32";
	        "MP101"."120VAC HEATER-2 POWER TR PRIMARY TRIPPED E6100CB" := "BA060AZSIMP101.33";
	        "MP101".SPARE_7 := "BA060AZSIMP101.34";
	        "MP101".SPARE_8 := "BA060AZSIMP101.35";
	        "MP101"."UPPER 2-1 HEATER POWER TRIPPED E6156CB" := "BA060AZSIMP101.36";
	        "MP101"."UPPER 2-2 HEATER POWER TRIPPED E6162CB" := "BA060AZSIMP101.37";
	       
	    END_REGION ;
	    REGION MP102
	        
	        "MP102"."LOWER 2-1 HEATER POWER TRIPPED E6168CB" := "BA060AZSIMP102.00";
	        "MP102"."LOWER 2-2 HEATER POWER TRIPPED E6174CB" := "BA060AZSIMP102.01";
	        "MP102"."LOWER 2-3 HEATER POWER TRIPPED E6180CB" := "BA060AZSIMP102.02";
	        "MP102"."VISION LIGHT CONTROLLER POWER STRIP OUTLET POWER TRIPPED E7184CB" := "BA060AZSIMP102.03";
	        "MP102"."120VAC CONTROL POWER TR PRIMARY TRIPPED E7100CB" := "BA060AZSIMP102.04";
	        "MP102"."120VAC CONTROL POWER TR SECONDARY TRIPPED E7110CB" := "BA060AZSIMP102.05";
	        "MP102"."CONTROL POWER ON TRIPPED E7116CB" := "BA060AZSIMP102.06";
	        "MP102"."MOTOR PANEL CONTROL POWER TRIPPED E7154CB" := "BA060AZSIMP102.07";
	        "MP102"."WEIGHT TESTER POWER STRIP OUTLET POWER TRIPPED E7160CB" := "BA060AZSIMP102.10";
	        "MP102"."VISION MONITOR & MCU POWER STRIP OUTLET POWER TRIPPED E7166CB" := "BA060AZSIMP102.11";
	        "MP102"."QR LASER MARKING TRIPPED E7172CB" := "BA060AZSIMP102.12";
	        "MP102"."HI-POT TESTER POWER STRIP OUTLET POWER TRIPPED E7178CB" := "BA060AZSIMP102.13";
	        "MP102"."FFU-1 POWER TRIPPED E7222CB" := "BA060AZSIMP102.14";
	        "MP102"."UPPER 1-1 TEMPERATURE CONTROLLER POWER TRIPPED E5206CB" := "BA060AZSIMP102.15";
	        "MP102"."UPPER 1-2 TEMPERATURE CONTROLLER POWER TRIPPED E5212CB" := "BA060AZSIMP102.16";
	        "MP102"."LOWER 1-1 TEMPERATURE CONTROLLER POWER TRIPPED E5218CB" := "BA060AZSIMP102.17";
	        "MP102"."LOWER 1-2 TEMPERATURE CONTROLLER POWER TRIPPED E5224CB" := "BA060AZSIMP102.20";
	        "MP102"."LOWER 1-3 TEMPERATURE CONTROLLER POWER TRIPPED E5230CB" := "BA060AZSIMP102.21";
	        "MP102"."UPPER 2-1 TEMPERATURE CONTROLLER POWER TRIPPED E6206CB" := "BA060AZSIMP102.22";
	        "MP102"."UPPER 2-2 TEMPERATURE CONTROLLER POWER TRIPPED E6212CB" := "BA060AZSIMP102.23";
	        "MP102"."LOWER 2-1 TEMPERATURE CONTROLLER POWER TRIPPED E6218CB" := "BA060AZSIMP102.24";
	        "MP102"."LOWER 2-2 TEMPERATURE CONTROLLER POWER TRIPPED E6224CB" := "BA060AZSIMP102.25";
	        "MP102"."LOWER 2-3 TEMPERATURE CONTROLLER POWER TRIPPED E6230CB" := "BA060AZSIMP102.26";
	        "MP102"."SPARE" := "BA060AZSIMP102.27";
	        "MP102"."CONTROL POWER SMPS DC OK E8104PWS" := "BA060AZSIMP102.30";
	        "MP102"."ET200MP I/O OUTPUT POWER TRIPPED E8154CB" := "BA060AZSIMP102.31";
	        "MP102"."JUNCTION BOX CONTROL POWER TRIPPED E8180CB" := "BA060AZSIMP102.32";
	        "MP102"."CLASS 2 SMPS POWER TRIPPED E8204CB" := "BA060AZSIMP102.33";
	        "MP102"."CLASS 2 SMPS MONITORING E8206PWS" := "BA060AZSIMP102.34";
	        "MP102"."ET200ECO PN-1 POWER TRIPPED E8220CB" := "BA060AZSIMP102.35";
	        "MP102"."ET200ECO PN-2 POWER TRIPPED E8224CB" := "BA060AZSIMP102.36";
	        "MP102"."ET200ECO PN-3 POWER TRIPPED E8228CB" := "BA060AZSIMP102.37";
	        
	    END_REGION ;
	    REGION MP103
	        "MP103"."ET200ECO PN-4 POWER TRIPPED E8232CB" := "BA060AZSIMP103.00";
	        "MP103"."PANEL FAN POWER TRIPPED E8304CB" := "BA060AZSIMP103.01";
	        "MP103"."SPARE" := "BA060AZSIMP103.02";
	        "MP103"."CONTROLLER POWER SMPS DC OK E8404PWS" := "BA060AZSIMP103.03";
	        "MP103"."CONTROLLER DC POWER TRIPPED E8406CB" := "BA060AZSIMP103.04";
	        "MP103"."KISTLER CONTROL POWER TRIPPED E8416CB" := "BA060AZSIMP103.05";
	        "MP103"."MANIFOLD-1 POWER TRIPPED E8422CB" := "BA060AZSIMP103.06";
	        "MP103"."MANIFOLD-2 POWER TRIPPED E8430CB" := "BA060AZSIMP103.07";
	        "MP103"."QR READER POWER TRIPPED E8456CB" := "BA060AZSIMP103.10";
	        "MP103"."QR READER POWER TRIPPED E8462CB" := "BA060AZSIMP103.11";
	        "MP103"."HANDY QR READER POWER TRIPPED E8468CB" := "BA060AZSIMP103.12";
	        "MP103"."PROFINET CONVERTER POWER TRIPPED E8474CB" := "BA060AZSIMP103.13";
	        "MP103"."MONITORING RELAY POWER TRIPPED E8504CB" := "BA060AZSIMP103.14";
	        "MP103"."SPARE" := "BA060AZSIMP103.15";
	        "MP103"."SAFETY POWER SMPS DC OK E8704PWS" := "BA060AZSIMP103.16";
	        "MP103"."SAFETY DC POWER TRIPPED E8706CB" := "BA060AZSIMP103.17";
	        "MP103"."ET200SP I/O SAFETY POWER TRIPPED E8716CB" := "BA060AZSIMP103.20";
	        "MP103"."JUNCTION BOX CONTROL POWER TRIPPED E8736CB" := "BA060AZSIMP103.21";
	        "MP103"."ET200ECO PN SAFETYT-1 POWER TRIPPED E8756CB" := "BA060AZSIMP103.22";
	        "MP103"."ET200ECO PN SAFETYT-2 POWER TRIPPED E8762CB" := "BA060AZSIMP103.23";
	        "MP103"."SPARE" := "BA060AZSIMP103.24";
	        "MP103"."CONTROL POWER SMPS DC OK E8804PWS" := "BA060AZSIMP103.25";
	        "MP103"."CONTROL DC POWER TRIPPED E8806CB" := "BA060AZSIMP103.26";
	        "MP103"."JUNCTION BOX CONTROL POWER TRIPPED E8816CB" := "BA060AZSIMP103.27";
	        "MP103"."DRIVE-CLIQ HUB POWER TRIPPED E8822CB" := "BA060AZSIMP103.30";
	        "MP103"."EQUIPMENT LED POWER TRIPPED E8828CB" := "BA060AZSIMP103.31";
	        // "MP103"."SPARE" := "BA060AZSIMP103.32";
	        // "MP103"."SPARE" := "BA060AZSIMP103.33";
	        // "MP103"."SPARE" := "BA060AZSIMP103.34";
	        // "MP103"."SPARE" := "BA060AZSIMP103.35";
	        // "MP103"."SPARE" := "BA060AZSIMP103.36";
	        // "MP103"."SPARE" := "BA060AZSIMP103.37";
	        
	        
	    END_REGION ;
	    REGION MP104
	        "MP104"."UPPER 1-1 HEATER MONITOR SIGNAL ON" := "BA060AZSIMP104.00";
	        "MP104"."UPPER 1-2 HEATER MONITOR SIGNAL ON" := "BA060AZSIMP104.01";
	        "MP104"."LOWER 1-1 HEATER MONITOR SIGNAL ON" := "BA060AZSIMP104.02";
	        "MP104"."LOWER 1-2 HEATER MONITOR SIGNAL ON" := "BA060AZSIMP104.03";
	        "MP104"."LOWER 1-3 HEATER MONITOR SIGNAL ON" := "BA060AZSIMP104.04";
	        "MP104"."UPPER 2-1 HEATER MONITOR SIGNAL ON" := "BA060AZSIMP104.05";
	        "MP104"."UPPER 2-2 HEATER MONITOR SIGNAL ON" := "BA060AZSIMP104.06";
	        "MP104"."LOWER 2-1 HEATER MONITOR SIGNAL ON" := "BA060AZSIMP104.07";
	        "MP104"."LOWER 2-2 HEATER MONITOR SIGNAL ON" := "BA060AZSIMP104.10";
	        "MP104"."LOWER 2-3 HEATER MONITOR SIGNAL ON" := "BA060AZSIMP104.11";
	        // "MP104"."SPARE" := "BA060AZSIMP104.12";
	        // "MP104"."SPARE_1" := "BA060AZSIMP104.13";
	        // "MP104"."SPARE_2" := "BA060AZSIMP104.14";
	        // "MP104"."SPARE_3" := "BA060AZSIMP104.15";
	        // "MP104"."SPARE_4" := "BA060AZSIMP104.16";
	        // "MP104"."SPARE_5" := "BA060AZSIMP104.17";
	        // "MP104"."SPARE_6" := "BA060AZSIMP104.20";
	        // "MP104"."SPARE_7" := "BA060AZSIMP104.21";
	        // "MP104"."SPARE_8" := "BA060AZSIMP104.22";
	        // "MP104"."SPARE_9" := "BA060AZSIMP104.23";
	        // "MP104"."SPARE_10" := "BA060AZSIMP104.24";
	        // "MP104"."SPARE_11" := "BA060AZSIMP104.25";
	        // "MP104"."SPARE_12" := "BA060AZSIMP104.26";
	        // "MP104"."SPARE_13" := "BA060AZSIMP104.27";
	        // "MP104"."SPARE_14" := "BA060AZSIMP104.30";
	        // "MP104"."SPARE_15" := "BA060AZSIMP104.31";
	        // "MP104"."SPARE_16" := "BA060AZSIMP104.32";
	        // "MP104"."SPARE_17" := "BA060AZSIMP104.33";
	        // "MP104"."SPARE_18" := "BA060AZSIMP104.34";
	        // "MP104"."SPARE_19" := "BA060AZSIMP104.35";
	        // "MP104"."SPARE_20" := "BA060AZSIMP104.36";
	        // "MP104"."SPARE_21" := "BA060AZSIMP104.37";
	        
	    END_REGION ;
	    REGION MP105
	        "MP105"."EQUIPMENT LED LAMP RELAY ON" := "BA060AZSIMP105.00";
	        // "MP105"."SPARE" := "BA060AZSIMP105.01";
	        // "MP105"."SPARE_1" := "BA060AZSIMP105.02";
	        "MP105"."CLASS2 SMPS ALARM RESET" := "BA060AZSIMP105.03";
	        // "MP105"."SPARE_2" := "BA060AZSIMP105.04";
	        // "MP105"."SPARE_3" := "BA060AZSIMP105.05";
	        // "MP105"."SPARE_4" := "BA060AZSIMP105.06";
	        // "MP105"."SPARE_5" := "BA060AZSIMP105.07";
	        "MP105"."QR MARKER TOWER LAMP 1 ON (RED)" := "BA060AZSIMP105.10";
	        "MP105"."QR MARKER TOWER LAMP 2 ON (AMBER)" := "BA060AZSIMP105.11";
	        "MP105"."QR MARKER TOWER LAMP 3 ON (GREEN)" := "BA060AZSIMP105.12";
	        "MP105"."QR MARKER TOWER LAMP 4 ON (WHITE)" := "BA060AZSIMP105.13";
	        "MP105"."QR MARKER TOWER LAMP 5 ON (BLUE)" := "BA060AZSIMP105.14";
	        "MP105"."QR MARKER TOWER LAMP BUZZER ON" := "BA060AZSIMP105.15";
	        // "MP105"."SPARE_6" := "BA060AZSIMP105.16";
	        // "MP105"."SPARE_7" := "BA060AZSIMP105.17";
	        // "MP105"."SPARE_8" := "BA060AZSIMP105.20";
	        // "MP105"."SPARE_9" := "BA060AZSIMP105.21";
	        // "MP105"."SPARE_10" := "BA060AZSIMP105.22";
	        // "MP105"."SPARE_11" := "BA060AZSIMP105.23";
	        // "MP105"."SPARE_12" := "BA060AZSIMP105.24";
	        // "MP105"."SPARE_13" := "BA060AZSIMP105.25";
	        // "MP105"."SPARE_14" := "BA060AZSIMP105.26";
	        // "MP105"."SPARE_15" := "BA060AZSIMP105.27";
	        // "MP105"."SPARE_16" := "BA060AZSIMP105.30";
	        // "MP105"."SPARE_17" := "BA060AZSIMP105.31";
	        // "MP105"."SPARE_18" := "BA060AZSIMP105.32";
	        // "MP105"."SPARE_19" := "BA060AZSIMP105.33";
	        // "MP105"."SPARE_20" := "BA060AZSIMP105.34";
	        // "MP105"."SPARE_21" := "BA060AZSIMP105.35";
	        // "MP105"."SPARE_22" := "BA060AZSIMP105.36";
	        // "MP105"."SPARE_23" := "BA060AZSIMP105.37";
	        
	    END_REGION ;
	    REGION MP106
	        "MP106"."MANIFOLD-1 SOL POWER MC FEEDBACK" := "BA060AZSISMP106.00";
	        "MP106"."MANIFOLD-2 SOL POWER MC FEEDBACK" := "BA060AZSISMP106.01";
	        "MP106"."QR LASER MARKING POWER 1 FEEDBACK" := "BA060AZSISMP106.02";
	        "MP106"."QR LASER MARKING POWER 2 FEEDBACK" := "BA060AZSISMP106.03";
	        "MP106"."FFU POWER MC 1 FEEDBACK" := "BA060AZSISMP106.04";
	        "MP106"."FFU POWER MC 2 FEEDBACK" := "BA060AZSISMP106.05";
	        "MP106"."SPARE" := "BA060AZSISMP106.06";
	        "MP106"."SPARE_1" := "BA060AZSISMP106.07";
	        "MP106"."SPARE_2" := "BA060AZSISMP106.10";
	        "MP106"."SPARE_3" := "BA060AZSISMP106.11";
	        "MP106"."SPARE_4" := "BA060AZSISMP106.12";
	        "MP106"."SPARE_5" := "BA060AZSISMP106.13";
	        "MP106"."SPARE_6" := "BA060AZSISMP106.14";
	        "MP106"."SPARE_7" := "BA060AZSISMP106.15";
	        "MP106"."SPARE_8" := "BA060AZSISMP106.16";
	        "MP106"."SPARE_9" := "BA060AZSISMP106.17";
	        "MP106".SPARE_20 := "BA060AZSISMP106.20";
	        "MP106".SPARE_21 := "BA060AZSISMP106.21";
	        "MP106".SPARE_22 := "BA060AZSISMP106.22";
	        "MP106".SPARE_23 := "BA060AZSISMP106.23";
	        "MP106".SPARE_24 := "BA060AZSISMP106.24";
	        "MP106".SPARE_25 := "BA060AZSISMP106.25";
	        "MP106"."SPARE_10" := "BA060AZSISMP106.26";
	        "MP106"."SPARE_11" := "BA060AZSISMP106.27";
	        "MP106"."SPARE_12" := "BA060AZSISMP106.30";
	        "MP106"."SPARE_13" := "BA060AZSISMP106.31";
	        "MP106"."SPARE_14" := "BA060AZSISMP106.32";
	        "MP106"."SPARE_15" := "BA060AZSISMP106.33";
	        "MP106"."SPARE_16" := "BA060AZSISMP106.34";
	        "MP106"."SPARE_17" := "BA060AZSISMP106.35";
	        "MP106"."SPARE_18" := "BA060AZSISMP106.37";
	        "MP106"."SPARE_19" := "BA060AZSISMP106.37";
	        
	    END_REGION ;
	    REGION MP107
	        "MP107"."MANIFOLD-1 SOL POWER MC ON" := "BA060AZSISMP107.00";
	        "MP107"."MANIFOLD-2 SOL POWER MC ON" := "BA060AZSISMP107.01";
	        "MP107"."QR LASER MARKING POWER ON 1" := "BA060AZSISMP107.02";
	        "MP107"."QR LASER MARKING POWER ON 2" := "BA060AZSISMP107.03";
	        "MP107"."FFU POWER MC ON 1" := "BA060AZSISMP107.04";
	        "MP107"."FFU POWER MC ON 2" := "BA060AZSISMP107.05";
	        "MP107"."SPARE" := "BA060AZSISMP107.06";
	        "MP107"."SPARE_1" := "BA060AZSISMP107.07";
	        
	    END_REGION ;
	    REGION MP108
	        "MP108"."10 TON SERVO PRESS-1 Z-AXIS EMS&STO SIGNAL" := "BA060AZSISMP108.00";
	        "MP108"."10 TON SERVO PRESS-1 Z-AXIS - PROBE 1" := "BA060AZSISMP108.01";
	        "MP108"."10 TON SERVO PRESS-2 Z-AXIS EMS&STO SIGNAL" := "BA060AZSISMP108.02";
	        "MP108"."10 TON SERVO PRESS-2 Z-AXIS - PROBE 1" := "BA060AZSISMP108.03";
	        "MP108"."3 TON SERVO PRESS Z-AXIS EMS&STO SIGNAL" := "BA060AZSISMP108.04";
	        "MP108"."3 TON SERVO PRESS Z-AXIS - PROBE 1" := "BA060AZSISMP108.05";
	        "MP108"."SPARE" := "BA060AZSISMP108.06";
	        "MP108"."SPARE_1" := "BA060AZSISMP108.07";
	        
	    END_REGION ;
	    REGION MP109
	        
	    END_REGION ;
	END_REGION
	REGION SP
	    REGION SP201
	        "SP201"."MAIN OP AUTO INITIATE PBL (GREEN)" := "BA060AZSISP201.00";
	        "SP201"."MAIN OP STOP PBL (RED)" := "BA060AZSISP201.01";
	        // "SP201"."RESERVE" := "BA060AZSISP201.02";
	        // "SP201"."SPARE" := "BA060AZSISP201.03";
	        // "SP201"."SPARE_1" := "BA060AZSISP201.04";
	        // "SP201"."SPARE_2" := "BA060AZSISP201.05";
	        // "SP201"."SPARE_3" := "BA060AZSISP201.06";
	        // "SP201"."SPARE_4" := "BA060AZSISP201.07";
	        "SP201"."MAIN HMI POWER TRIPPED E110CB" := "BA060AZSISP201.10";
	        // "SP201"."SPARE_5" := "BA060AZSISP201.11";
	        // "SP201"."SPARE_6" := "BA060AZSISP201.12";
	        // "SP201"."SPARE_7" := "BA060AZSISP201.13";
	        // "SP201"."SPARE_8" := "BA060AZSISP201.14";
	        // "SP201"."SPARE_9" := "BA060AZSISP201.15";
	        // "SP201"."SPARE_10" := "BA060AZSISP201.16";
	        // "SP201"."SPARE_11" := "BA060AZSISP201.17";
	        
	    END_REGION ;
	    REGION SP202
	        "SP202"."MAIN OP AUTO INITIATE PBL LAMP ON (GREEN)" := "BA060AZSISP202.00";
	        "SP202"."MAIN OP STOP PBL LAMP ON (RED)" := "BA060AZSISP202.01";
	        "SP202"."RESERVE" := "BA060AZSISP202.02";
	        "SP202"."MAIN OP ENABLE PBL LAMP ON (WHITE)" := "BA060AZSISP202.03";
	        "SP202"."MAIN OP SAFETY RESET PBL LAMP ON (BLUE)" := "BA060AZSISP202.04";
	        "SP202"."SPARE" := "BA060AZSISP202.05";
	        "SP202"."SPARE_1" := "BA060AZSISP202.06";
	        "SP202"."SPARE_2" := "BA060AZSISP202.07";
	        "SP202"."TOWER LAMP 1 ON (RED)" := "BA060AZSISP202.10";
	        "SP202"."TOWER LAMP 2 ON (AMBER)" := "BA060AZSISP202.11";
	        "SP202"."TOWER LAMP 3 ON (GREEN)" := "BA060AZSISP202.12";
	        "SP202"."TOWER LAMP 4 ON (WHITE)" := "BA060AZSISP202.13";
	        "SP202"."TOWER LAMP 5 ON (BLUE)" := "BA060AZSISP202.14";
	        "SP202"."TOWER LAMP BUZZER ON" := "BA060AZSISP202.15";
	        "SP202"."SPARE_3" := "BA060AZSISP202.16";
	        "SP202"."SPARE_4" := "BA060AZSISP202.17";
	        
	    END_REGION ;
	    REGION SP203
	        "SP203"."MAIN OP MODE SLELECT SS.AUTO" := "BA060AZSISP203.00";
	        "SP203"."MAIN OP HOME PBL (GREEN)" := "BA060AZSISP203.01";
	        "SP203"."MAIN OP SAFETY RESET PBL (BLUE)" := "BA060AZSISP203.02";
	        "SP203"."MAIN OP SCS MODE SLELECT SS.AUTO" := "BA060AZSISP203.03";
	        "SP203"."MAIN OP MODE SLELECT SS.MANUAL" := "BA060AZSISP203.04";
	        "SP203"."MAIN OP ENABLE PBL (WHITE)" := "BA060AZSISP203.05";
	        "SP203"."MAIN OP SCS MODE SLELECT SS.SETUP" := "BA060AZSISP203.06";
	        "SP203"."MAIN OP SCS MODE SLELECT SS.DISABLE" := "BA060AZSISP203.07";
	        
	    END_REGION ;
	    REGION SP204
	        "SP204"."MAIN OP EMERGENCY STOP CH.A" := "BA060AZSISP204.00";
	        "SP204"."SPARE" := "BA060AZSISP204.01";
	        "SP204"."SPARE_1" := "BA060AZSISP204.02";
	        "SP204"."SPARE_2" := "BA060AZSISP204.03";
	        "SP204"."MAIN OP EMERGENCY STOP CH.B" := "BA060AZSISP204.04";
	        "SP204"."SPARE_3" := "BA060AZSISP204.05";
	        "SP204"."SPARE_4" := "BA060AZSISP204.06";
	        "SP204"."SPARE_5" := "BA060AZSISP204.07";
	        
	    END_REGION ;
	    REGION SP205
	        "SP205"."MAIN OP PENDANT REQUIRED PL LAMP ON (YELLOW)" := "BA060AZSISP205.00";
	        "SP205"."SPARE" := "BA060AZSISP205.01";
	        "SP205"."MAIN OP HOME PBL LAMP ON (GREEN)" := "BA060AZSISP205.02";
	        "SP205"."SPARE_1" := "BA060AZSISP205.03";
	        "SP205"."SPARE_2" := "BA060AZSISP205.04";
	        "SP205"."SPARE_3" := "BA060AZSISP205.05";
	        "SP205"."SPARE_4" := "BA060AZSISP205.06";
	        "SP205"."MAIN OP SCS MODE SELECT DISABLE PL LAMP ON (GREEN)" := "BA060AZSISP205.07";
	        
	    END_REGION ;
	    REGION SP501
	        "SP501"."SPARE" := "BA060AZSISP501.00";
	        "SP501"."SAFETY DC POWER TRIPPED E218CB" := "BA060AZSISP501.01";
	        "SP501"."CLASS 2 SMPS POWER TRIPPED E308CB" := "BA060AZSISP501.02";
	        "SP501"."CLASS 2 SMPS MONITORING E310PWS" := "BA060AZSISP501.03";
	        "SP501"."ET200ECO PN-1 POWER TRIPPED E324CB" := "BA060AZSISP501.04";
	        "SP501"."ET200ECO PN-2 POWER TRIPPED E328CB" := "BA060AZSISP501.05";
	        "SP501"."ET200ECO PN-3 POWER TRIPPED E332CB" := "BA060AZSISP501.06";
	        "SP501"."ET200ECO PN-4 POWER TRIPPED E336CB" := "BA060AZSISP501.07";
	        "SP501".SPARE_1 := "BA060AZSISP501.10";
	        "SP501".SPARE_2 := "BA060AZSISP501.11";
	        "SP501".SPARE_3 := "BA060AZSISP501.12";
	        "SP501".SPARE_4 := "BA060AZSISP501.13";
	        "SP501".SPARE_5 := "BA060AZSISP501.14";
	        "SP501".SPARE_6 := "BA060AZSISP501.15";
	        "SP501".SPARE_7 := "BA060AZSISP501.16";
	        "SP501".SPARE_8 := "BA060AZSISP501.17";
	        
	    END_REGION ;
	    REGION SP502
	        "SP502"."UPPER 1-1 HEATER TEMPERATURE CONTROLLER ALARM" := "BA060AZSISP502.00";
	        "SP502"."SPARE" := "BA060AZSISP502.01";
	        "SP502"."UPPER 1-2 HEATER TEMPERATURE CONTROLLER ALARM" := "BA060AZSISP502.02";
	        "SP502"."SPARE_1" := "BA060AZSISP502.03";
	        "SP502"."LOWER 1-1 HEATER TEMPERATURE CONTROLLER ALARM" := "BA060AZSISP502.04";
	        "SP502"."SPARE_2" := "BA060AZSISP502.05";
	        "SP502"."LOWER 1-2 HEATER TEMPERATURE CONTROLLER ALARM" := "BA060AZSISP502.06";
	        "SP502"."SPARE_3" := "BA060AZSISP502.07";
	        "SP502"."LOWER 1-3 HEATER TEMPERATURE CONTROLLER ALARM" := "BA060AZSISP502.10";
	        // "SP502"."SPARE_4" := "BA060AZSISP502.11";
	        // "SP502"."SPARE_5" := "BA060AZSISP502.12";
	        // "SP502"."SPARE_6" := "BA060AZSISP502.13";
	        // "SP502"."SPARE_7" := "BA060AZSISP502.14";
	        // "SP502"."SPARE_8" := "BA060AZSISP502.15";
	        "SP502"."VISION BUSY (STO)" := "BA060AZSISP502.16";
	        "SP502"."VISION RESULT (OK)" := "BA060AZSISP502.17";
	        
	    END_REGION ;
	    REGION SP503
	        "SP503"."UPPER 2-1 HEATER TEMPERATURE CONTROLLER ALARM" := "BA060AZSISP503.00";
	        "SP503"."SPARE" := "BA060AZSISP503.01";
	        "SP503"."UPPER 2-2 HEATER TEMPERATURE CONTROLLER ALARM" := "BA060AZSISP503.02";
	        "SP503"."SPARE_1" := "BA060AZSISP503.03";
	        "SP503"."LOWER 2-1 HEATER TEMPERATURE CONTROLLER ALARM" := "BA060AZSISP503.04";
	        "SP503"."SPARE_2" := "BA060AZSISP503.05";
	        "SP503"."LOWER 2-2 HEATER TEMPERATURE CONTROLLER ALARM" := "BA060AZSISP503.06";
	        "SP503"."SPARE_3" := "BA060AZSISP503.07";
	        "SP503"."LOWER 2-3 HEATER TEMPERATURE CONTROLLER ALARM" := "BA060AZSISP503.10";
	        "SP503"."SPARE_4" := "BA060AZSISP503.11";
	        // "SP503"."SPARE_5" := "BA060AZSISP503.12";
	        // "SP503"."SPARE_6" := "BA060AZSISP503.13";
	        // "SP503"."SPARE_7" := "BA060AZSISP503.14";
	        // "SP503"."SPARE_8" := "BA060AZSISP503.15";
	        "SP503"."STACK-1 LIGHT CURTAIN STATUS/SELECT" := "BA060AZSISP503.16";
	        "SP503"."STACK-2 LIGHT CURTAIN STATUS/SELECT" := "BA060AZSISP503.17";
	        
	    END_REGION ;
	    REGION SP504
	        "SP504"."CLASS2 SMPS ALARM RESET" := "BA060AZSISP504.00";
	        "SP504"."SPARE" := "BA060AZSISP504.01";
	        "SP504"."VISION CONTROLLER TRIGGER IN" := "BA060AZSISP504.02";
	        "SP504"."SPARE_1" := "BA060AZSISP504.03";
	        "SP504"."QR MARKING TRIGGER IN" := "BA060AZSISP504.04";
	        "SP504"."SPARE_2" := "BA060AZSISP504.05";
	        "SP504"."SPARE_3" := "BA060AZSISP504.06";
	        "SP504"."SPARE_4" := "BA060AZSISP504.07";
	        "SP504".SPARE_5 := "BA060AZSISP504.10";
	        "SP504".SPARE_6 := "BA060AZSISP504.11";
	        "SP504".SPARE_7 := "BA060AZSISP504.12";
	        "SP504".SPARE_8 := "BA060AZSISP504.13";
	        "SP504".SPARE_9 := "BA060AZSISP504.14";
	        "SP504".SPARE_10 := "BA060AZSISP504.15";
	        "SP504".SPARE_11 := "BA060AZSISP504.16";
	        "SP504".SPARE_12 := "BA060AZSISP504.17";
	        
	    END_REGION ;
	    REGION SP505
	        "SP505".SPARE := "BA060AZSISP505.00";
	        "SP505"."SPARE_1" := "BA060AZSISP505.01";
	        "SP505".SPARE_2 := "BA060AZSISP505.02";
	        "SP505"."SPARE_3" := "BA060AZSISP505.03";
	        "SP505".SPARE_4 := "BA060AZSISP505.04";
	        "SP505"."SPARE_5" := "BA060AZSISP505.05";
	        "SP505".SPARE_6 := "BA060AZSISP505.06";
	        "SP505"."SPARE_7" := "BA060AZSISP505.07";
	        "SP505".SPARE_8 := "BA060AZSISP505.10";
	        // "SP505"."SPARE_4" := "BA060AZSISP505.11";
	        // "SP505"."SPARE_5" := "BA060AZSISP505.12";
	        // "SP505"."SPARE_6" := "BA060AZSISP505.13";
	        // "SP505"."SPARE_7" := "BA060AZSISP505.14";
	        // "SP505"."SPARE_8" := "BA060AZSISP505.15";
	        // "SP505"."SPARE_9" := "BA060AZSISP505.16";
	        // "SP505"."SPARE_10" := "BA060AZSISP505.17";
	        
	    END_REGION ;
	    REGION SP506
	        "SP506".SPARE := "BA060AZSISP506.00";
	        "SP506"."SPARE_1" := "BA060AZSISP506.01";
	        "SP506".SPARE_2 := "BA060AZSISP506.02";
	        "SP506"."SPARE_3" := "BA060AZSISP506.03";
	        "SP506".SPARE_4 := "BA060AZSISP506.04";
	        "SP506"."SPARE_5" := "BA060AZSISP506.05";
	        "SP506".SPARE_6 := "BA060AZSISP506.06";
	        "SP506"."SPARE_7" := "BA060AZSISP506.07";
	        "SP506".SPARE_8 := "BA060AZSISP506.10";
	        // "SP506"."SPARE_4" := "BA060AZSISP506.11";
	        // "SP506"."SPARE_5" := "BA060AZSISP506.12";
	        // "SP506"."SPARE_6" := "BA060AZSISP506.13";
	        // "SP506"."SPARE_7" := "BA060AZSISP506.14";
	        // "SP506"."SPARE_8" := "BA060AZSISP506.15";
	        "SP506"."STACK-1 LIGHT CURTAIN RESET" := "BA060AZSISP506.16";
	        "SP506"."STACK-2 LIGHT CURTAIN RESET" := "BA060AZSISP506.17";
	        
	    END_REGION ;
	    REGION SP507
	        "SP507"."PHMI-1 EMERGENCY STOP CH.A" := "BA060AZSISP507.00";
	        "SP507"."PHMI-1 ENABLE SWITCH CH.A" := "BA060AZSISP507.01";
	        "SP507"."PHMI-2 EMERGENCY STOP CH.A" := "BA060AZSISP507.02";
	        "SP507"."PHMI-2 ENABLE SWITCH CH.A" := "BA060AZSISP507.03";
	        "SP507"."PHMI-1 EMERGENCY STOP CH.B" := "BA060AZSISP507.04";
	        "SP507"."PHMI-1 ENABLE SWITCH CH.B" := "BA060AZSISP507.05";
	        "SP507"."PHMI-2 EMERGENCY STOP CH.B" := "BA060AZSISP507.06";
	        "SP507"."PHMI-2 ENABLE SWITCH CH.B" := "BA060AZSISP507.07";
	        
	    END_REGION ;
	    REGION SP508
	        "SP508"."STACK-1 LIGHT CURTAIN OSSD 1" := "BA060AZSISP508.00";
	        "SP508"."STACK-2 LIGHT CURTAIN OSSD 1" := "BA060AZSISP508.01";
	        "SP508"."QR MARKING SHUTTER STATUS OUTPUT" := "BA060AZSISP508.02";
	        "SP508"."SPARE" := "BA060AZSISP508.03";
	        "SP508"."STACK-1 LIGHT CURTAIN OSSD 2" := "BA060AZSISP508.04";
	        "SP508"."STACK-2 LIGHT CURTAIN OSSD 2" := "BA060AZSISP508.05";
	        "SP508"."SPARE_1" := "BA060AZSISP508.06";
	        "SP508"."SPARE_2" := "BA060AZSISP508.07";
	//        "SP508"."Value Status Of STACK-1 LIGHT CURTAIN OSSD1" := "BA060AZSISP508.10";
	//        "SP508"."Value Status Of STACK-1 LIGHT CURTAIN OSSD2" := "BA060AZSISP508.14";
	        
	    END_REGION ;
	    REGION SP509
	        "SP509"."QR MARKING SHUTTER CONTROL INPUT A" := "BA060AZSISP509.00";
	        "SP509"."QR MARKING SHUTTER CONTROL INPUT B" := "BA060AZSISP509.01";
	        "SP509"."SPARE" := "BA060AZSISP509.02";
	        "SP509"."SPARE_1" := "BA060AZSISP509.03";
	        "SP509"."SPARE_2" := "BA060AZSISP509.04";
	        "SP509"."SPARE_3" := "BA060AZSISP509.05";
	        "SP509"."SPARE_4" := "BA060AZSISP509.06";
	        "SP509"."SPARE_5" := "BA060AZSISP509.07";
	        
	    END_REGION ;
	REGION "SP510"
	        // "SP510"."HI-POT TESTER SERIAL COMMUNICATION":="BA060AZSISP510.00"
	        // "SP510"."SPARE":="BA060AZSISP510.01"
	        // "SP510"."SPARE_1":="BA060AZSISP510.02"
	        // "SP510"."SPARE_2":="BA060AZSISP510.03"
	        // "SP510"."SPARE_3":="BA060AZSISP510.04"
	        // "SP510"."SPARE_4":="BA060AZSISP510.05"
	        // "SP510"."SPARE_5":="BA060AZSISP510.06"
	        // "SP510"."SPARE_6":="BA060AZSISP510.07"
	        // "SP510"."SPARE_7":="BA060AZSISP510.10"
	        // "SP510"."SPARE_8":="BA060AZSISP510.11"
	        // "SP510"."SPARE_9":="BA060AZSISP510.12"
	        // "SP510"."SPARE_10":="BA060AZSISP510.13"
	        // "SP510"."SPARE_11":="BA060AZSISP510.14"
	        // "SP510"."SPARE_12":="BA060AZSISP510.15"
	        // "SP510"."SPARE_13":="BA060AZSISP510.16"
	        // "SP510"."SPARE_14":="BA060AZSISP510.17"
	        
	    END_REGION ;
	    REGION SP511
	        // "SP511"."SPARE":="BA060AZSISP511.00"
	        // "SP511"."SPARE_1":="BA060AZSISP511.01"
	        // "SP511"."SPARE_2":="BA060AZSISP511.02"
	        // "SP511"."SPARE_3":="BA060AZSISP511.03"
	        // "SP511"."SPARE_5":="BA060AZSISP511.04"
	        // "SP511"."SPARE_6":="BA060AZSISP511.05"
	        // "SP511"."SPARE_7":="BA060AZSISP511.06"
	        // "SP511"."SPARE_9":="BA060AZSISP511.07"
	        // "SP511"."HEATER-1 TEMPERATURE CONTROLLER RS485":="BA060AZSISP511.10"
	        // "SP511"."SPARE_10":="BA060AZSISP511.11"
	        // "SP511"."SPARE_11":="BA060AZSISP511.12"
	        // "SP511"."SPARE_12":="BA060AZSISP511.13"
	        // "SP511"."SPARE_13":="BA060AZSISP511.14"
	        // "SP511"."SPARE_14":="BA060AZSISP511.15"
	        
	    END_REGION ;
	    REGION SP512
	 //     "SP512"."SPARE":="BA060AZSISP512.00"
	 //     "SP512"."SPARE_1":="BA060AZSISP512.01"
	 //       "SP512"."SPARE_2":="BA060AZSISP512.02"
	 //       "SP512"."SPARE_3":="BA060AZSISP512.03"
	 //       "SP512"."SPARE_4":="BA060AZSISP512.04"
	 //       "SP512"."SPARE_5":="BA060AZSISP512.05"
	 //       "SP512"."SPARE_6":="BA060AZSISP512.06"
	 //       "SP512"."SPARE_7":="BA060AZSISP512.07"
	 //       "SP512"."SPARE_8":="BA060AZSISP512.10"
	 //       "SP512"."SPARE_9":="BA060AZSISP512.11"
	 //       "SP512"."HEATER-2 TEMPERATURE CONTROLLER RS485":="BA060AZSISP512.12"
	 //       "SP512"."SPARE_10":="BA060AZSISP512.13"
	 //       "SP512"."SPARE_11":="BA060AZSISP512.14"
	 //       "SP512"."SPARE_12":="BA060AZSISP512.15"
	 //       "SP512"."SPARE_13":="BA060AZSISP512.16"
	 //       "SP512"."SPARE_14":="BA060AZSISP512.17"
	        
	    END_REGION ;
	END_REGION ;
	        
	        
	        
	        
	        
END_FUNCTION

FUNCTION "CallProductionData" : Void   // FC151, LAD
TITLE = Production data
AUTHOR : SICAR
FAMILY : ProdData
VERSION : 1.0
// Call of  FC ProductDataSimulation and LSicar Production Blocks
// stored: IsIECCheckEnabled true, SetENOAutomatically true
   // Ret_Val : Ret_Val
   VAR_TEMP   // added for the SCL form of the ladder/FBD networks
      _w1 : Bool;
      _w2 : Bool;
      _w3 : Bool;
      _w4 : Bool;
      _w5 : Bool;
      _w6 : Bool;
      _w7 : Bool;
      _w8 : Bool;
      _w9 : Bool;
      _w10 : Bool;
   END_VAR
BEGIN

REGION Network 1: BLOCK INFO HEADER
   // SIEMENS AG / (c)Copyright 2023
   // ------------------------------------------------------------------------------
   // Title:            CallProductionData(FC151)
   // Comment/Function: Call of  FC ProductDataSimulation and LSicar Production Blocks
   // Library/Family:   Automation Framework
   // Author:           Siemens Digital Industry
   // Tested with:      ---
   // Engineering:      TIA Portal V19
   // Restrictions:     -
   // Requirements:     ---
   // ------------------------------------------------------------------------------
   // Change log table:
   // Version  | Date       | Expert in charge       | Changes applied
   // ---------|------------|------------------------|------------------------------
   // 01.00.00 | 11.12.2023 | Siemens Industry Online Support
   //                         First released version
END_REGION

